C07280=1077.683,437.352,387.565,177.005,33.132,155.992
C07281=1077.692,437.598,387.519,177.011,33.146,155.996
C07282=1077.700,437.843,387.473,177.017,33.159,155.999
C07283=1077.707,438.089,387.426,177.024,33.173,156.002
C07284=1077.715,438.334,387.380,177.031,33.186,156.005
C07285=1077.726,438.676,387.315,177.040,33.205,156.010
C07286=1077.738,439.018,387.250,177.048,33.224,156.014
C07287=1077.749,439.359,387.186,177.058,33.243,156.019
C07288=1077.761,439.701,387.121,177.067,33.262,156.023
C07289=1077.771,440.033,387.057,177.077,33.281,156.028
C07290=1077.782,440.366,386.995,177.085,33.300,156.032
C07291=1077.793,440.699,386.931,177.094,33.319,156.037
C07292=1077.804,441.033,386.867,177.104,33.338,156.041
C07293=1077.812,441.277,386.821,177.110,33.352,156.045
C07294=1077.820,441.523,386.774,177.118,33.366,156.048
C07295=1077.829,441.768,386.726,177.124,33.380,156.052
C07296=1077.837,442.014,386.679,177.130,33.395,156.055
C07297=1077.845,442.259,386.633,177.138,33.409,156.059
C07298=1077.853,442.504,386.584,177.144,33.423,156.062
C07299=1077.861,442.749,386.538,177.152,33.438,156.065
C07300=1077.869,442.995,386.490,177.158,33.452,156.069
C07301=1077.877,443.239,386.443,177.166,33.467,156.072
C07302=1077.885,443.485,386.396,177.173,33.482,156.076
C07303=1077.894,443.730,386.349,177.179,33.496,156.080
C07304=1077.902,443.976,386.301,177.187,33.511,156.083
C07305=1077.911,444.221,386.254,177.193,33.525,156.087
C07306=1077.919,444.467,386.206,177.201,33.540,156.090
C07307=1077.927,444.712,386.158,177.208,33.555,156.094
C07308=1077.935,444.957,386.111,177.215,33.570,156.097
C07309=1077.944,445.202,386.063,177.222,33.585,156.101
C07310=1077.952,445.447,386.015,177.229,33.600,156.105
C07311=1077.960,445.693,385.968,177.237,33.615,156.108
C07312=1077.968,445.938,385.920,177.244,33.630,156.112
C07313=1077.976,446.183,385.872,177.252,33.645,156.116
C07314=1077.985,446.428,385.825,177.258,33.660,156.119
C07315=1077.993,446.673,385.777,177.265,33.675,156.123
C07316=1078.002,446.918,385.729,177.271,33.690,156.127
C07317=1078.010,447.164,385.681,177.278,33.706,156.131
C07318=1078.019,447.408,385.632,177.285,33.721,156.134
C07319=1078.027,447.653,385.584,177.290,33.736,156.138
C07320=1078.035,447.898,385.536,177.296,33.751,156.142
C07321=1078.043,448.143,385.488,177.302,33.766,156.146
C07322=1078.052,448.388,385.440,177.306,33.781,156.149
C07323=1078.061,448.634,385.392,177.311,33.796,156.153
C07324=1078.069,448.878,385.343,177.316,33.811,156.157
C07325=1078.079,449.123,385.296,177.320,33.826,156.161
C07326=1078.090,449.368,385.249,177.325,33.840,156.164
C07327=1078.102,449.613,385.203,177.329,33.853,156.168
C07328=1078.116,449.859,385.158,177.333,33.866,156.171
C07329=1077.755,449.854,384.928,177.311,34.027,156.213
C07330=1077.741,449.608,384.974,177.306,34.015,156.210
C07331=1077.728,449.363,385.020,177.302,34.001,156.207
C07332=1077.716,449.117,385.067,177.298,33.987,156.203
C07333=1077.707,448.873,385.113,177.293,33.973,156.200
C07334=1077.698,448.628,385.162,177.288,33.958,156.196
C07335=1077.690,448.383,385.210,177.283,33.942,156.192
C07336=1077.681,448.139,385.258,177.277,33.927,156.188
C07337=1077.673,447.894,385.306,177.272,33.912,156.185
C07338=1077.664,447.649,385.355,177.266,33.897,156.181
C07339=1077.656,447.403,385.404,177.260,33.882,156.177
C07340=1077.647,447.158,385.451,177.253,33.867,156.173
C07341=1077.639,446.913,385.499,177.248,33.852,156.170
C07342=1077.631,446.668,385.547,177.240,33.836,156.166
C07343=1077.622,446.423,385.596,177.233,33.821,156.162
C07344=1077.613,446.178,385.643,177.226,33.806,156.158
C07345=1077.605,445.933,385.691,177.219,33.791,156.155
C07346=1077.597,445.688,385.739,177.211,33.776,156.151
C07347=1077.589,445.443,385.787,177.204,33.761,156.147
C07348=1077.580,445.198,385.835,177.197,33.746,156.144
C07349=1077.572,444.952,385.882,177.189,33.731,156.140
C07350=1077.564,444.707,385.930,177.182,33.716,156.136
C07351=1077.555,444.462,385.978,177.175,33.701,156.133
C07352=1077.547,444.217,386.026,177.168,33.686,156.129
C07353=1077.539,443.971,386.072,177.161,33.672,156.126
C07354=1077.531,443.726,386.120,177.153,33.657,156.122
C07355=1077.522,443.481,386.168,177.146,33.643,156.118
C07356=1077.514,443.235,386.215,177.139,33.628,156.115
C07357=1077.506,442.990,386.263,177.132,33.613,156.111
C07358=1077.497,442.745,386.310,177.125,33.599,156.108
C07359=1077.490,442.500,386.358,177.118,33.585,156.104
C07360=1077.481,442.255,386.404,177.111,33.570,156.101
C07361=1077.474,442.009,386.452,177.104,33.556,156.097
C07362=1077.465,441.764,386.499,177.097,33.542,156.094
C07363=1077.457,441.519,386.546,177.090,33.527,156.091
C07364=1077.449,441.273,386.593,177.083,33.513,156.087
C07365=1077.440,441.028,386.640,177.077,33.499,156.084
C07366=1077.430,440.712,386.700,177.067,33.481,156.079
C07367=1077.420,440.397,386.761,177.059,33.463,156.075
C07368=1077.409,440.080,386.821,177.050,33.445,156.071
C07369=1077.399,439.764,386.881,177.042,33.427,156.067
C07370=1077.391,439.519,386.928,177.034,33.413,156.063
C07371=1077.383,439.274,386.975,177.028,33.399,156.060
C07372=1077.375,439.029,387.021,177.022,33.386,156.057
C07373=1077.367,438.783,387.067,177.014,33.372,156.053
C07374=1077.358,438.537,387.114,177.008,33.359,156.050
C07375=1077.350,438.292,387.161,177.002,33.345,156.047
C07376=1077.342,438.046,387.207,176.994,33.332,156.044
C07377=1077.334,437.801,387.253,176.988,33.318,156.040
C07378=1077.326,437.555,387.300,176.982,33.305,156.037
C07379=1077.319,437.310,387.346,176.975,33.291,156.034
C07380=1077.310,437.065,387.393,176.968,33.278,156.031
C07381=1077.302,436.819,387.438,176.962,33.265,156.028
C07382=1077.294,436.574,387.485,176.955,33.251,156.025
C07383=1077.286,436.328,387.531,176.949,33.238,156.021
C07384=1077.278,436.082,387.577,176.943,33.225,156.018
C07385=1077.270,435.837,387.623,176.936,33.212,156.015
C07386=1077.262,435.592,387.669,176.929,33.199,156.012
C07387=1077.254,435.346,387.715,176.923,33.186,156.009
C07388=1077.246,435.101,387.761,176.917,33.173,156.006
C07389=1077.239,434.855,387.807,176.911,33.160,156.003
C07390=1077.230,434.609,387.853,176.904,33.147,156.000
C07391=1077.223,434.364,387.898,176.898,33.134,155.997
C07392=1077.215,434.118,387.944,176.892,33.121,155.994
C07393=1077.207,433.872,387.990,176.886,33.108,155.991
C07394=1077.200,433.627,388.036,176.880,33.095,155.988
C07395=1077.192,433.381,388.082,176.872,33.083,155.985
C07396=1077.184,433.136,388.127,176.866,33.070,155.982
C07397=1077.176,432.891,388.173,176.860,33.058,155.979
C07398=1077.168,432.644,388.219,176.854,33.045,155.976
C07399=1077.161,432.398,388.264,176.848,33.032,155.973
C07400=1077.153,432.153,388.309,176.842,33.020,155.970
C07401=1077.145,431.907,388.355,176.835,33.007,155.967
C07402=1077.138,431.662,388.401,176.829,32.995,155.964
C07403=1077.130,431.416,388.445,176.824,32.982,155.961
C07404=1077.122,431.170,388.491,176.818,32.970,155.958
C07405=1077.114,430.924,388.536,176.812,32.958,155.956
C07406=1077.107,430.679,388.581,176.806,32.946,155.953
C07407=1077.099,430.433,388.626,176.800,32.933,155.950
C07408=1077.091,430.187,388.671,176.794,32.921,155.947
C07409=1077.083,429.941,388.716,176.788,32.909,155.944
C07410=1077.076,429.696,388.762,176.781,32.897,155.941
C07411=1077.069,429.450,388.807,176.775,32.885,155.939
C07412=1077.060,429.204,388.851,176.769,32.873,155.936
C07413=1077.053,428.959,388.897,176.763,32.861,155.933
C07414=1077.045,428.713,388.942,176.758,32.849,155.930
C07415=1077.037,428.467,388.986,176.752,32.837,155.928
C07416=1077.030,428.221,389.031,176.746,32.825,155.925
C07417=1077.023,427.975,389.076,176.740,32.813,155.922
C07418=1077.013,427.678,389.130,176.733,32.799,155.919
C07419=1077.004,427.380,389.184,176.726,32.785,155.916
C07420=1076.994,427.083,389.238,176.719,32.770,155.912
C07421=1076.986,426.787,389.292,176.712,32.756,155.909
C07422=1076.978,426.571,389.331,176.707,32.747,155.907
C07423=1076.972,426.356,389.370,176.702,32.737,155.904
C07424=1076.965,426.141,389.409,176.697,32.726,155.902
C07425=1076.959,425.925,389.447,176.692,32.716,155.900
C07426=1076.951,425.680,389.492,176.686,32.705,155.897
C07427=1076.944,425.433,389.537,176.681,32.693,155.894
C07428=1076.936,425.188,389.581,176.675,32.682,155.892
C07429=1076.929,424.941,389.625,176.669,32.671,155.889
C07430=1076.921,424.696,389.669,176.664,32.659,155.887
C07431=1076.913,424.450,389.713,176.658,32.648,155.884
C07432=1076.906,424.204,389.758,176.652,32.637,155.881
C07433=1076.898,423.958,389.802,176.647,32.625,155.879
C07434=1076.892,423.712,389.846,176.641,32.614,155.876
C07435=1076.884,423.466,389.890,176.635,32.603,155.874
C07436=1076.876,423.220,389.934,176.630,32.592,155.871
C07437=1076.869,422.974,389.978,176.625,32.581,155.869
C07438=1076.861,422.728,390.022,176.620,32.569,155.866
C07439=1076.854,422.482,390.067,176.614,32.559,155.864
C07440=1076.847,422.236,390.110,176.608,32.547,155.861
C07441=1076.839,421.990,390.154,176.603,32.536,155.859
C07442=1076.832,421.745,390.198,176.597,32.525,155.856
C07443=1076.825,421.498,390.242,176.592,32.515,155.854
C07444=1076.817,421.252,390.286,176.586,32.504,155.851
C07445=1076.810,421.006,390.329,176.581,32.493,155.849
C07446=1076.802,420.760,390.372,176.575,32.482,155.846
C07447=1076.794,420.513,390.416,176.570,32.472,155.844
C07448=1076.787,420.268,390.459,176.565,32.461,155.841
C07449=1076.780,420.021,390.504,176.560,32.450,155.839
C07450=1076.773,419.775,390.547,176.554,32.439,155.837
C07451=1076.765,419.529,390.590,176.549,32.428,155.834
C07452=1076.758,419.283,390.634,176.543,32.418,155.832
C07453=1076.750,419.037,390.677,176.538,32.408,155.830
C07454=1076.743,418.791,390.721,176.532,32.397,155.827
C07455=1076.735,418.545,390.764,176.528,32.386,155.825
C07456=1076.728,418.299,390.807,176.522,32.376,155.822
C07457=1076.720,418.053,390.851,176.517,32.366,155.820
C07458=1076.713,417.807,390.894,176.512,32.355,155.818
C07459=1076.706,417.561,390.937,176.506,32.345,155.815
C07460=1076.698,417.315,390.980,176.501,32.334,155.813
C07461=1076.692,417.068,391.023,176.496,32.324,155.811
C07462=1076.684,416.822,391.067,176.491,32.314,155.808
C07463=1076.677,416.576,391.110,176.486,32.303,155.806
C07464=1076.670,416.330,391.152,176.480,32.293,155.804
C07465=1076.662,416.084,391.196,176.475,32.283,155.802
C07466=1076.655,415.837,391.239,176.470,32.272,155.799
C07467=1076.648,415.592,391.282,176.465,32.262,155.797
C07468=1076.641,415.346,391.324,176.460,32.252,155.795
C07469=1076.634,415.099,391.367,176.455,32.242,155.792
C07470=1076.627,414.853,391.411,176.449,32.232,155.790
C07471=1076.619,414.607,391.452,176.444,32.222,155.788
C07472=1076.611,414.360,391.495,176.440,32.212,155.786
C07473=1076.604,414.114,391.539,176.435,32.203,155.784
C07474=1076.597,413.868,391.581,176.429,32.193,155.781
C07475=1076.589,413.621,391.623,176.424,32.183,155.779
C07476=1076.582,413.375,391.666,176.420,32.173,155.777
C07477=1076.576,413.129,391.709,176.414,32.163,155.775
C07478=1076.569,412.880,391.752,176.409,32.153,155.773
C07479=1076.560,412.631,391.795,176.404,32.143,155.770
C07480=1076.553,412.382,391.838,176.399,32.133,155.768
C07481=1076.546,412.132,391.881,176.394,32.123,155.766
C07482=1076.539,411.886,391.923,176.389,32.114,155.764
C07483=1076.531,411.640,391.965,176.384,32.104,155.762
C07484=1076.525,411.394,392.008,176.379,32.094,155.760
C07485=1076.518,411.148,392.050,176.375,32.085,155.758
C07486=1076.510,410.902,392.092,176.369,32.075,155.755
C07487=1076.503,410.655,392.135,176.364,32.065,155.753
C07488=1076.496,410.409,392.177,176.359,32.056,155.751
C07489=1076.489,410.162,392.218,176.355,32.047,155.749
C07490=1076.482,409.915,392.261,176.350,32.037,155.747
C07491=1076.474,409.669,392.303,176.345,32.027,155.745
C07492=1076.467,409.423,392.346,176.341,32.018,155.743
C07493=1076.461,409.176,392.388,176.336,32.008,155.741
C07494=1076.453,408.930,392.430,176.330,31.999,155.739
C07495=1076.447,408.685,392.472,176.325,31.989,155.737
C07496=1076.440,408.438,392.513,176.321,31.981,155.735
C07497=1076.433,408.192,392.556,176.316,31.971,155.733
C07498=1076.425,407.946,392.597,176.311,31.962,155.731
C07499=1076.419,407.699,392.639,176.307,31.952,155.729
C07500=1076.412,407.453,392.682,176.302,31.943,155.727
C07501=1076.404,407.206,392.723,176.297,31.934,155.725
C07502=1076.398,406.959,392.765,176.292,31.925,155.723
C07503=1076.390,406.713,392.807,176.288,31.915,155.721
C07504=1076.384,406.466,392.849,176.283,31.907,155.719
C07505=1076.376,406.220,392.891,176.278,31.897,155.717
C07506=1076.369,405.974,392.931,176.274,31.888,155.715
C07507=1076.363,405.727,392.973,176.269,31.879,155.713
C07508=1076.356,405.481,393.015,176.264,31.870,155.711
C07509=1076.348,405.235,393.056,176.260,31.861,155.709
C07510=1076.341,404.988,393.098,176.255,31.852,155.707
C07511=1076.334,404.741,393.140,176.250,31.843,155.705
C07512=1076.327,404.496,393.180,176.246,31.834,155.703
C07513=1076.321,404.249,393.222,176.241,31.825,155.701
C07514=1076.313,404.003,393.264,176.236,31.817,155.699
C07515=1076.306,403.756,393.305,176.232,31.808,155.697
C07516=1076.300,403.510,393.347,176.227,31.799,155.695
C07517=1076.293,403.263,393.388,176.222,31.790,155.693
C07518=1076.286,403.017,393.429,176.219,31.781,155.691
C07519=1076.278,402.770,393.471,176.214,31.772,155.690
C07520=1076.272,402.524,393.511,176.209,31.764,155.688
C07521=1076.265,402.277,393.552,176.205,31.755,155.686
C07522=1076.257,402.030,393.593,176.200,31.746,155.684
C07523=1076.251,401.784,393.635,176.195,31.738,155.682
C07524=1076.244,401.538,393.676,176.191,31.729,155.680
C07525=1076.237,401.291,393.717,176.186,31.720,155.678
C07526=1076.230,401.045,393.758,176.181,31.712,155.677
C07527=1076.223,400.798,393.798,176.178,31.703,155.675
C07528=1076.216,400.551,393.840,176.173,31.695,155.673
C07529=1076.209,400.305,393.881,176.168,31.686,155.671
C07530=1076.202,400.059,393.922,176.164,31.678,155.669
C07531=1076.195,399.812,393.962,176.159,31.669,155.667
C07532=1076.188,399.566,394.003,176.154,31.661,155.666
C07533=1076.181,399.320,394.044,176.151,31.652,155.664
C07534=1076.175,399.074,394.085,176.146,31.644,155.662
C07535=1076.168,398.827,394.125,176.142,31.635,155.660
C07536=1076.161,398.581,394.166,176.137,31.627,155.658
C07537=1076.155,398.334,394.206,176.132,31.619,155.657
C07538=1076.147,398.088,394.248,176.129,31.611,155.655
C07539=1076.141,397.841,394.288,176.124,31.602,155.653
C07540=1076.134,397.595,394.329,176.119,31.594,155.651
C07541=1076.127,397.348,394.369,176.115,31.586,155.650
C07542=1076.119,397.102,394.410,176.111,31.578,155.648
C07543=1076.113,396.855,394.450,176.107,31.569,155.646
C07544=1076.106,396.608,394.490,176.102,31.561,155.644
C07545=1076.099,396.362,394.531,176.097,31.553,155.643
C07546=1076.092,396.115,394.572,176.094,31.545,155.641
C07547=1076.086,395.868,394.612,176.089,31.537,155.639
C07548=1076.079,395.622,394.651,176.084,31.528,155.638
C07549=1076.072,395.376,394.693,176.080,31.520,155.636
C07550=1076.065,395.129,394.733,176.076,31.512,155.634
C07551=1076.059,394.883,394.773,176.072,31.504,155.632
C07552=1076.052,394.635,394.814,176.067,31.496,155.631
C07553=1076.045,394.389,394.853,176.063,31.489,155.629
C07554=1076.038,394.143,394.893,176.059,31.481,155.627
C07555=1076.031,393.895,394.934,176.054,31.472,155.626
C07556=1076.025,393.649,394.974,176.050,31.464,155.624
C07557=1076.018,393.403,395.013,176.046,31.457,155.622
C07558=1076.011,393.155,395.054,176.041,31.449,155.621
C07559=1076.004,392.909,395.094,176.037,31.441,155.619
C07560=1075.997,392.663,395.134,176.033,31.433,155.617
C07561=1075.991,392.416,395.174,176.029,31.425,155.616
C07562=1075.983,392.169,395.214,176.024,31.417,155.614
C07563=1075.977,391.923,395.254,176.020,31.409,155.612
C07564=1075.971,391.676,395.294,176.016,31.402,155.611
C07565=1075.963,391.430,395.334,176.011,31.394,155.609
C07566=1075.957,391.183,395.373,176.008,31.386,155.608
C07567=1075.950,390.936,395.413,176.003,31.378,155.606
C07568=1075.943,390.690,395.453,175.999,31.371,155.604
C07569=1075.936,390.443,395.493,175.995,31.363,155.603
C07570=1075.930,390.196,395.532,175.990,31.355,155.601
C07571=1075.923,389.950,395.572,175.986,31.348,155.600
C07572=1075.915,389.702,395.611,175.982,31.340,155.598
C07573=1075.909,389.456,395.651,175.978,31.332,155.596
C07574=1075.902,389.210,395.691,175.974,31.325,155.595
C07575=1075.896,388.963,395.730,175.970,31.317,155.593
C07576=1075.889,388.716,395.769,175.965,31.310,155.592
C07577=1075.882,388.470,395.808,175.961,31.302,155.590
C07578=1075.876,388.223,395.848,175.957,31.295,155.589
C07579=1075.869,387.976,395.887,175.953,31.287,155.587
C07580=1075.862,387.730,395.927,175.949,31.280,155.586
C07581=1075.856,387.483,395.966,175.944,31.272,155.584
C07582=1075.848,387.237,396.006,175.941,31.265,155.583
C07583=1075.841,386.989,396.045,175.936,31.257,155.581
C07584=1075.835,386.742,396.084,175.932,31.250,155.579
C07585=1075.828,386.496,396.124,175.928,31.243,155.578
C07586=1075.822,386.257,396.161,175.924,31.236,155.576
C07587=1075.816,386.018,396.200,175.920,31.228,155.575
C07588=1075.809,385.779,396.237,175.916,31.222,155.574
C07589=1075.803,385.540,396.275,175.913,31.214,155.572
C07590=1075.796,385.301,396.314,175.908,31.207,155.571
C07591=1075.790,385.062,396.352,175.904,31.200,155.569
C07592=1075.784,384.824,396.389,175.900,31.193,155.568
C07593=1075.777,384.585,396.427,175.896,31.186,155.566
C07594=1075.770,384.338,396.466,175.893,31.179,155.565
C07595=1075.764,384.091,396.505,175.888,31.171,155.563
C07596=1075.757,383.844,396.545,175.885,31.164,155.562
C07597=1075.751,383.598,396.583,175.880,31.157,155.560
C07598=1075.744,383.351,396.622,175.876,31.150,155.559
C07599=1075.738,383.104,396.661,175.872,31.142,155.557
C07600=1075.731,382.857,396.700,175.868,31.135,155.556
C07601=1075.724,382.611,396.739,175.864,31.128,155.555
C07602=1075.717,382.364,396.778,175.860,31.121,155.553
C07603=1075.711,382.117,396.817,175.856,31.114,155.552
C07604=1075.705,381.870,396.855,175.852,31.107,155.550
C07605=1075.699,381.623,396.894,175.848,31.100,155.549
C07606=1075.692,381.376,396.933,175.844,31.093,155.547
C07607=1075.685,381.129,396.972,175.840,31.086,155.546
C07608=1075.678,380.883,397.011,175.836,31.079,155.544
C07609=1075.672,380.635,397.049,175.831,31.072,155.543
C07610=1075.665,380.389,397.087,175.828,31.065,155.542
C07611=1075.659,380.142,397.126,175.824,31.058,155.540
C07612=1075.652,379.895,397.165,175.820,31.051,155.539
C07613=1075.645,379.648,397.203,175.816,31.044,155.537
C07614=1075.638,379.401,397.241,175.812,31.037,155.536
C07615=1075.632,379.155,397.280,175.808,31.030,155.535
C07616=1075.625,378.908,397.318,175.804,31.023,155.533
C07617=1075.618,378.661,397.357,175.800,31.016,155.532
C07618=1075.612,378.414,397.395,175.797,31.010,155.531
C07619=1075.606,378.168,397.433,175.792,31.003,155.529
C07620=1075.599,377.920,397.471,175.789,30.996,155.528
C07621=1075.592,377.673,397.510,175.784,30.989,155.526
C07622=1075.586,377.426,397.548,175.781,30.982,155.525
C07623=1075.579,377.180,397.587,175.777,30.975,155.524
C07624=1075.573,376.932,397.625,175.772,30.969,155.522
C07625=1075.566,376.686,397.663,175.769,30.962,155.521
C07626=1075.560,376.439,397.701,175.765,30.955,155.520
C07627=1075.553,376.192,397.739,175.761,30.948,155.518
C07628=1075.547,375.945,397.777,175.757,30.942,155.517
C07629=1075.540,375.698,397.816,175.754,30.935,155.516
C07630=1075.534,375.450,397.854,175.749,30.928,155.514
C07631=1075.528,375.204,397.892,175.746,30.922,155.513
C07632=1075.521,374.957,397.930,175.741,30.915,155.511
C07633=1075.514,374.711,397.967,175.738,30.908,155.510
C07634=1075.508,374.463,398.006,175.734,30.902,155.509
C07635=1075.502,374.217,398.044,175.730,30.895,155.507
C07636=1075.495,373.969,398.082,175.726,30.888,155.506
C07637=1075.489,373.722,398.120,175.723,30.882,155.505
C07638=1075.483,373.475,398.158,175.719,30.875,155.504
C07639=1075.476,373.228,398.196,175.715,30.869,155.502
C07640=1075.470,372.981,398.233,175.711,30.862,155.501
C07641=1075.462,372.734,398.271,175.708,30.856,155.500
C07642=1075.456,372.510,398.306,175.704,30.850,155.499
C07643=1075.451,372.285,398.340,175.700,30.844,155.497
C07644=1075.445,372.062,398.374,175.697,30.838,155.496
C07645=1075.439,371.837,398.408,175.693,30.832,155.495
C07646=1075.433,371.612,398.443,175.690,30.826,155.494
C07647=1075.427,371.388,398.476,175.686,30.820,155.493
C07648=1075.421,371.164,398.511,175.683,30.815,155.492
C07649=1075.416,370.939,398.545,175.679,30.809,155.490
C07650=1075.408,370.692,398.582,175.676,30.802,155.489
C07651=1075.402,370.445,398.620,175.672,30.796,155.488
C07652=1075.395,370.198,398.657,175.668,30.790,155.487
C07653=1075.390,369.951,398.695,175.664,30.783,155.485
C07654=1075.383,369.704,398.733,175.660,30.777,155.484
C07655=1075.376,369.457,398.770,175.657,30.770,155.483
C07656=1075.370,369.210,398.808,175.652,30.764,155.482
C07657=1075.364,368.963,398.844,175.649,30.758,155.480
C07658=1075.358,368.716,398.882,175.645,30.752,155.479
C07659=1075.350,368.469,398.920,175.642,30.745,155.478
C07660=1075.345,368.221,398.957,175.638,30.739,155.477
C07661=1075.338,367.974,398.994,175.634,30.733,155.476
C07662=1075.332,367.727,399.032,175.630,30.726,155.474
C07663=1075.325,367.480,399.068,175.627,30.720,155.473
C07664=1075.318,367.233,399.106,175.623,30.714,155.472
C07665=1075.313,366.986,399.143,175.619,30.708,155.471
C07666=1075.306,366.740,399.180,175.615,30.701,155.469
C07667=1075.300,366.491,399.218,175.612,30.695,155.468
C07668=1075.293,366.245,399.255,175.608,30.689,155.467
C07669=1075.287,365.998,399.292,175.605,30.683,155.466
C07670=1075.280,365.750,399.329,175.600,30.677,155.465
C07671=1075.275,365.503,399.366,175.597,30.671,155.463
C07672=1075.268,365.257,399.403,175.593,30.664,155.462
C07673=1075.262,365.010,399.440,175.590,30.658,155.461
C07674=1075.255,364.762,399.477,175.586,30.652,155.460
C07675=1075.249,364.515,399.514,175.582,30.646,155.459
C07676=1075.242,364.268,399.551,175.578,30.640,155.457
C07677=1075.236,364.020,399.588,175.575,30.634,155.456
C07678=1075.230,363.773,399.625,175.571,30.628,155.455
C07679=1075.223,363.527,399.662,175.568,30.622,155.454
C07680=1075.217,363.279,399.698,175.564,30.616,155.453
C07681=1075.210,363.032,399.735,175.560,30.610,155.452
C07682=1075.204,362.784,399.772,175.556,30.604,155.450
C07683=1075.198,362.537,399.809,175.553,30.598,155.449
C07684=1075.191,362.291,399.846,175.549,30.592,155.448
C07685=1075.184,362.043,399.883,175.546,30.586,155.447
C07686=1075.178,361.796,399.919,175.542,30.580,155.446
C07687=1075.172,361.549,399.956,175.539,30.574,155.445
C07688=1075.165,361.302,399.992,175.534,30.568,155.444
C07689=1075.160,361.055,400.029,175.531,30.562,155.442
C07690=1075.153,360.807,400.066,175.527,30.556,155.441
C07691=1075.147,360.560,400.102,175.524,30.550,155.440
C07692=1075.140,360.313,400.139,175.520,30.545,155.439
C07693=1075.134,360.066,400.175,175.517,30.539,155.438
C07694=1075.128,359.819,400.212,175.513,30.533,155.437
C07695=1075.121,359.572,400.248,175.510,30.527,155.436
C07696=1075.115,359.325,400.285,175.505,30.521,155.435
C07697=1075.108,359.076,400.321,175.502,30.515,155.433
C07698=1075.103,358.861,400.352,175.499,30.510,155.432
C07699=1075.097,358.645,400.384,175.496,30.505,155.431
C07700=1075.092,358.428,400.416,175.493,30.500,155.430
C07701=1075.086,358.212,400.448,175.490,30.495,155.430
C07702=1075.080,357.996,400.480,175.486,30.490,155.429
C07703=1075.075,357.780,400.511,175.483,30.485,155.428
C07704=1075.070,357.564,400.543,175.480,30.480,155.427
C07705=1075.064,357.348,400.575,175.477,30.475,155.426
C07706=1075.057,357.101,400.611,175.474,30.469,155.425
C07707=1075.051,356.853,400.647,175.470,30.463,155.423
C07708=1075.045,356.606,400.683,175.466,30.457,155.422
C07709=1075.039,356.359,400.720,175.462,30.452,155.421
C07710=1075.033,356.111,400.756,175.459,30.446,155.420
C07711=1075.026,355.864,400.792,175.455,30.440,155.419
C07712=1075.020,355.617,400.828,175.452,30.434,155.418
C07713=1075.014,355.369,400.864,175.448,30.429,155.417
C07714=1075.008,355.122,400.901,175.445,30.423,155.416
C07715=1075.002,354.875,400.936,175.441,30.417,155.415
C07716=1074.995,354.628,400.972,175.438,30.412,155.414
C07717=1074.989,354.380,401.008,175.434,30.406,155.413
C07718=1074.982,354.133,401.044,175.431,30.401,155.412
C07719=1074.976,353.886,401.080,175.427,30.395,155.411
C07720=1074.970,353.638,401.116,175.424,30.389,155.409
C07721=1074.964,353.391,401.152,175.420,30.384,155.408
C07722=1074.958,353.143,401.188,175.417,30.378,155.407
C07723=1074.951,352.896,401.224,175.413,30.372,155.406
C07724=1074.945,352.649,401.260,175.410,30.367,155.405
C07725=1074.939,352.401,401.295,175.406,30.361,155.404
C07726=1074.932,352.154,401.332,175.403,30.356,155.403
C07727=1074.926,351.907,401.367,175.400,30.350,155.402
C07728=1074.920,351.659,401.403,175.396,30.345,155.401
C07729=1074.913,351.411,401.438,175.393,30.339,155.400
C07730=1074.906,351.165,401.474,175.389,30.334,155.399
C07731=1074.901,350.918,401.510,175.386,30.328,155.398
C07732=1074.895,350.670,401.545,175.382,30.323,155.397
C07733=1074.888,350.423,401.580,175.379,30.317,155.396
C07734=1074.882,350.175,401.616,175.375,30.312,155.395
C07735=1074.876,349.927,401.652,175.372,30.306,155.394
C07736=1074.869,349.681,401.688,175.368,30.301,155.393
C07737=1074.863,349.433,401.723,175.365,30.296,155.392
C07738=1074.856,349.185,401.759,175.361,30.290,155.391
C07739=1074.851,348.938,401.794,175.358,30.285,155.390
C07740=1074.845,348.691,401.830,175.354,30.279,155.389
C07741=1074.838,348.443,401.865,175.351,30.274,155.388
C07742=1074.832,348.196,401.901,175.347,30.269,155.387
C07743=1074.825,347.948,401.936,175.344,30.263,155.386
C07744=1074.820,347.701,401.971,175.340,30.258,155.385
C07745=1074.813,347.454,402.006,175.337,30.252,155.384
C07746=1074.807,347.206,402.042,175.333,30.247,155.383
C07747=1074.801,346.958,402.076,175.330,30.242,155.382
C07748=1074.795,346.711,402.112,175.326,30.236,155.381
C07749=1074.789,346.464,402.147,175.323,30.231,155.380
C07750=1074.782,346.216,402.183,175.320,30.226,155.379
C07751=1074.776,345.969,402.218,175.317,30.220,155.378
C07752=1074.770,345.721,402.253,175.313,30.215,155.377
C07753=1074.763,345.475,402.288,175.310,30.210,155.376
C07754=1074.758,345.260,402.318,175.306,30.205,155.375
C07755=1074.753,345.045,402.349,175.304,30.200,155.374
C07756=1074.748,344.831,402.379,175.301,30.196,155.373
C07757=1074.742,344.616,402.410,175.298,30.191,155.373
C07758=1074.737,344.402,402.441,175.295,30.187,155.372
C07759=1074.731,344.188,402.471,175.293,30.182,155.371
C07760=1074.726,343.974,402.501,175.289,30.178,155.370
C07761=1074.721,343.759,402.531,175.286,30.173,155.369
C07762=1074.714,343.511,402.566,175.283,30.168,155.368
C07763=1074.708,343.265,402.601,175.279,30.163,155.367
C07764=1074.702,343.016,402.636,175.276,30.158,155.366
C07765=1074.695,342.769,402.671,175.273,30.152,155.365
C07766=1074.690,342.522,402.705,175.269,30.147,155.364
C07767=1074.684,342.274,402.741,175.266,30.142,155.363
C07768=1074.677,342.026,402.775,175.263,30.137,155.362
C07769=1074.671,341.779,402.810,175.260,30.132,155.362
C07770=1074.664,341.531,402.845,175.256,30.126,155.361
C07771=1074.658,341.284,402.880,175.253,30.121,155.360
C07772=1074.653,341.036,402.914,175.249,30.116,155.359
C07773=1074.646,340.789,402.950,175.246,30.111,155.358
C07774=1074.640,340.542,402.984,175.242,30.105,155.357
C07775=1074.634,340.294,403.019,175.239,30.100,155.356
C07776=1074.627,340.046,403.054,175.236,30.096,155.355
C07777=1074.622,339.799,403.088,175.233,30.091,155.354
C07778=1074.615,339.551,403.123,175.229,30.085,155.353
C07779=1074.609,339.304,403.157,175.226,30.080,155.352
C07780=1074.603,339.056,403.192,175.222,30.075,155.351
C07781=1074.597,338.808,403.226,175.219,30.070,155.350
C07782=1074.591,338.561,403.261,175.216,30.065,155.349
C07783=1074.585,338.314,403.295,175.213,30.060,155.348
C07784=1074.578,338.066,403.330,175.209,30.055,155.348
C07785=1074.573,337.818,403.364,175.206,30.049,155.347
C07786=1074.566,337.571,403.399,175.202,30.044,155.346
C07787=1074.560,337.323,403.434,175.200,30.040,155.345
C07788=1074.554,337.076,403.468,175.196,30.035,155.344
C07789=1074.548,336.828,403.502,175.193,30.030,155.343
C07790=1074.542,336.580,403.536,175.189,30.024,155.342
C07791=1074.535,336.332,403.571,175.186,30.019,155.341
C07792=1074.529,336.085,403.605,175.183,30.014,155.340
C07793=1074.523,335.837,403.639,175.180,30.010,155.339
C07794=1074.517,335.590,403.673,175.177,30.004,155.338
C07795=1074.511,335.342,403.708,175.173,29.999,155.338
C07796=1074.504,335.095,403.742,175.170,29.994,155.337
C07797=1074.498,334.847,403.776,175.167,29.990,155.336
C07798=1074.492,334.600,403.810,175.164,29.985,155.335
C07799=1074.486,334.352,403.844,175.160,29.980,155.334
C07800=1074.479,334.104,403.878,175.157,29.975,155.333
C07801=1074.474,333.857,403.912,175.153,29.970,155.332
C07802=1074.467,333.609,403.947,175.151,29.965,155.331
C07803=1074.461,333.362,403.981,175.147,29.960,155.330
C07804=1074.455,333.114,404.015,175.144,29.955,155.330
C07805=1074.449,332.866,404.049,175.140,29.950,155.329
C07806=1074.443,332.619,404.083,175.138,29.946,155.328
C07807=1074.437,332.371,404.117,175.134,29.940,155.327
C07808=1074.431,332.123,404.151,175.131,29.935,155.326
C07809=1074.425,331.876,404.185,175.127,29.930,155.325
C07810=1074.419,331.659,404.215,175.125,29.926,155.324
C07811=1074.414,331.443,404.244,175.122,29.922,155.324
C07812=1074.408,331.225,404.274,175.120,29.918,155.323
C07813=1074.403,331.009,404.303,175.116,29.913,155.322
C07814=1074.398,330.791,404.334,175.114,29.910,155.321
C07815=1074.392,330.573,404.363,175.111,29.905,155.321
C07816=1074.387,330.357,404.393,175.108,29.901,155.320
C07817=1074.381,330.140,404.422,175.105,29.897,155.319
C07818=1074.375,329.892,404.455,175.102,29.892,155.318
C07819=1074.369,329.644,404.490,175.099,29.888,155.318
C07820=1074.362,329.397,404.522,175.096,29.882,155.317
C07821=1074.356,329.150,404.556,175.092,29.878,155.316
C07822=1074.350,328.902,404.591,175.090,29.873,155.315
C07823=1074.344,328.654,404.624,175.086,29.868,155.314
C07824=1074.338,328.407,404.658,175.083,29.863,155.313
C07825=1074.331,328.158,404.691,175.079,29.859,155.312
C07826=1074.325,327.911,404.725,175.077,29.854,155.312
C07827=1074.319,327.663,404.758,175.073,29.849,155.311
C07828=1074.312,327.415,404.792,175.070,29.844,155.310
C07829=1074.306,327.168,404.825,175.067,29.840,155.309
C07830=1074.300,326.920,404.858,175.064,29.835,155.308
C07831=1074.295,326.673,404.892,175.060,29.830,155.307
C07832=1074.288,326.424,404.925,175.057,29.826,155.307
C07833=1074.282,326.177,404.959,175.054,29.821,155.306
C07834=1074.276,325.930,404.992,175.051,29.816,155.305
C07835=1074.270,325.682,405.025,175.047,29.811,155.304
C07836=1074.263,325.434,405.059,175.045,29.807,155.303
C07837=1074.257,325.186,405.092,175.041,29.802,155.303
C07838=1074.251,324.938,405.125,175.038,29.797,155.302
C07839=1074.245,324.691,405.159,175.035,29.793,155.301
C07840=1074.239,324.444,405.192,175.032,29.788,155.300
C07841=1074.233,324.195,405.226,175.028,29.783,155.299
C07842=1074.226,323.947,405.258,175.026,29.779,155.298
C07843=1074.221,323.699,405.292,175.022,29.774,155.298
C07844=1074.214,323.453,405.325,175.020,29.770,155.297
C07845=1074.209,323.205,405.359,175.017,29.765,155.296
C07846=1074.202,322.957,405.391,175.013,29.760,155.295
C07847=1074.196,322.709,405.424,175.011,29.756,155.294
C07848=1074.190,322.462,405.457,175.007,29.751,155.293
C07849=1074.184,322.213,405.491,175.004,29.746,155.293
C07850=1074.178,321.965,405.524,175.001,29.742,155.292
C07851=1074.172,321.718,405.557,174.998,29.737,155.291
C07852=1074.166,321.470,405.591,174.994,29.732,155.290
C07853=1074.160,321.223,405.623,174.992,29.728,155.289
C07854=1074.153,320.975,405.656,174.988,29.723,155.289
C07855=1074.148,320.727,405.689,174.986,29.719,155.288
C07856=1074.141,320.480,405.722,174.982,29.714,155.287
C07857=1074.136,320.232,405.756,174.979,29.709,155.286
C07858=1074.130,319.984,405.788,174.976,29.705,155.285
C07859=1074.124,319.736,405.822,174.973,29.700,155.285
C07860=1074.118,319.488,405.854,174.970,29.696,155.284
C07861=1074.112,319.241,405.886,174.967,29.691,155.283
C07862=1074.106,318.993,405.920,174.964,29.686,155.282
C07863=1074.100,318.745,405.953,174.961,29.682,155.281
C07864=1074.094,318.497,405.985,174.958,29.677,155.281
C07865=1074.088,318.250,406.019,174.955,29.673,155.280
C07866=1074.083,318.030,406.047,174.952,29.668,155.279
C07867=1074.078,317.809,406.077,174.949,29.664,155.278
C07868=1074.072,317.589,406.106,174.946,29.660,155.278
C07869=1074.067,317.369,406.135,174.944,29.656,155.277
C07870=1074.062,317.149,406.165,174.941,29.652,155.276
C07871=1074.057,316.929,406.194,174.939,29.648,155.275
C07872=1074.051,316.708,406.223,174.935,29.644,155.275
C07873=1074.046,316.488,406.251,174.933,29.640,155.274
C07874=1074.040,316.240,406.284,174.930,29.636,155.273
C07875=1074.034,315.993,406.317,174.927,29.630,155.272
C07876=1074.028,315.745,406.349,174.924,29.626,155.272
C07877=1074.022,315.497,406.382,174.921,29.622,155.271
C07878=1074.016,315.249,406.415,174.918,29.617,155.270
C07879=1074.011,315.002,406.447,174.915,29.613,155.269
C07880=1074.005,314.754,406.480,174.912,29.608,155.269
C07881=1073.999,314.506,406.513,174.909,29.604,155.268
C07882=1073.993,314.258,406.545,174.906,29.599,155.267
C07883=1073.987,314.010,406.578,174.903,29.595,155.266
C07884=1073.981,313.762,406.610,174.900,29.590,155.265
C07885=1073.974,313.514,406.642,174.897,29.586,155.265
C07886=1073.968,313.266,406.674,174.894,29.581,155.264
C07887=1073.961,313.019,406.706,174.890,29.577,155.263
C07888=1073.955,312.771,406.738,174.888,29.573,155.262
C07889=1073.949,312.523,406.771,174.884,29.568,155.262
C07890=1073.943,312.275,406.803,174.882,29.564,155.261
C07891=1073.937,312.028,406.836,174.878,29.560,155.260
C07892=1073.931,311.780,406.868,174.876,29.555,155.259
C07893=1073.925,311.532,406.900,174.872,29.551,155.259
C07894=1073.918,311.284,406.932,174.870,29.546,155.258
C07895=1073.912,311.036,406.964,174.866,29.542,155.257
C07896=1073.906,310.789,406.997,174.864,29.538,155.256
C07897=1073.901,310.541,407.028,174.861,29.533,155.256
C07898=1073.895,310.293,407.060,174.858,29.529,155.255
C07899=1073.888,310.045,407.092,174.855,29.525,155.254
C07900=1073.882,309.797,407.124,174.851,29.520,155.253
C07901=1073.876,309.549,407.156,174.849,29.516,155.253
C07902=1073.870,309.301,407.189,174.845,29.511,155.252
C07903=1073.864,309.054,407.221,174.843,29.507,155.251
C07904=1073.857,308.806,407.252,174.839,29.503,155.251
C07905=1073.851,308.558,407.284,174.837,29.498,155.250
C07906=1073.845,308.310,407.316,174.833,29.494,155.249
C07907=1073.840,308.062,407.348,174.831,29.490,155.248
C07908=1073.834,307.815,407.381,174.827,29.485,155.248
C07909=1073.827,307.567,407.412,174.825,29.481,155.247
C07910=1073.822,307.319,407.444,174.821,29.477,155.246
C07911=1073.816,307.071,407.476,174.819,29.472,155.245
C07912=1073.810,306.823,407.508,174.815,29.468,155.245
C07913=1073.803,306.576,407.539,174.813,29.464,155.244
C07914=1073.797,306.327,407.571,174.810,29.459,155.243
C07915=1073.791,306.079,407.603,174.807,29.455,155.242
C07916=1073.786,305.832,407.635,174.804,29.451,155.242
C07917=1073.779,305.584,407.667,174.801,29.446,155.241
C07918=1073.773,305.336,407.699,174.799,29.442,155.240
C07919=1073.768,305.089,407.731,174.795,29.438,155.240
C07920=1073.761,304.841,407.762,174.793,29.433,155.239
C07921=1073.755,304.592,407.794,174.789,29.429,155.238
C07922=1073.751,304.374,407.821,174.787,29.425,155.237
C07923=1073.746,304.155,407.849,174.784,29.421,155.237
C07924=1073.740,303.937,407.877,174.782,29.418,155.236
C07925=1073.735,303.718,407.905,174.779,29.414,155.235
C07926=1073.729,303.500,407.933,174.777,29.410,155.235
C07927=1073.724,303.281,407.961,174.774,29.406,155.234
C07928=1073.719,303.063,407.989,174.772,29.402,155.233
C07929=1073.714,302.844,408.017,174.769,29.398,155.233
C07930=1073.708,302.597,408.048,174.766,29.394,155.232
C07931=1073.701,302.349,408.080,174.763,29.390,155.231
C07932=1073.696,302.101,408.112,174.760,29.385,155.231
C07933=1073.690,301.852,408.143,174.757,29.381,155.230
C07934=1073.684,301.605,408.174,174.755,29.377,155.229
C07935=1073.678,301.357,408.206,174.751,29.373,155.229
C07936=1073.672,301.110,408.237,174.749,29.368,155.228
C07937=1073.666,300.861,408.269,174.745,29.364,155.227
C07938=1073.661,300.613,408.300,174.743,29.360,155.226
C07939=1073.654,300.365,408.331,174.739,29.355,155.226
C07940=1073.649,300.118,408.363,174.737,29.351,155.225
C07941=1073.643,299.869,408.394,174.734,29.347,155.224
C07942=1073.637,299.622,408.426,174.731,29.342,155.223
C07943=1073.631,299.374,408.458,174.729,29.339,155.223
C07944=1073.626,299.126,408.488,174.725,29.334,155.222
C07945=1073.620,298.878,408.520,174.723,29.329,155.221
C07946=1073.614,298.630,408.552,174.720,29.326,155.220
C07947=1073.608,298.382,408.582,174.717,29.321,155.220
C07948=1073.602,298.134,408.614,174.714,29.317,155.219
C07949=1073.596,297.886,408.644,174.711,29.312,155.218
C07950=1073.591,297.639,408.676,174.708,29.308,155.218
C07951=1073.585,297.390,408.707,174.706,29.304,155.217
C07952=1073.579,297.143,408.738,174.702,29.299,155.216
C07953=1073.573,296.894,408.769,174.700,29.296,155.215
C07954=1073.567,296.647,408.801,174.697,29.291,155.215
C07955=1073.561,296.398,408.831,174.694,29.287,155.214
C07956=1073.555,296.151,408.862,174.692,29.283,155.213
C07957=1073.549,295.902,408.894,174.688,29.279,155.213
C07958=1073.543,295.654,408.924,174.686,29.275,155.212
C07959=1073.537,295.407,408.955,174.683,29.271,155.211
C07960=1073.532,295.158,408.987,174.680,29.266,155.211
C07961=1073.525,294.911,409.018,174.677,29.262,155.210
C07962=1073.519,294.663,409.048,174.674,29.258,155.209
C07963=1073.513,294.415,409.079,174.671,29.254,155.208
C07964=1073.508,294.167,409.110,174.669,29.250,155.208
C07965=1073.501,293.919,409.141,174.665,29.245,155.207
C07966=1073.496,293.671,409.171,174.663,29.241,155.206
C07967=1073.489,293.422,409.202,174.660,29.237,155.206
C07968=1073.483,293.175,409.233,174.657,29.233,155.205
C07969=1073.478,292.927,409.264,174.655,29.229,155.204
C07970=1073.472,292.678,409.295,174.652,29.225,155.204
C07971=1073.466,292.431,409.325,174.649,29.220,155.203
C07972=1073.460,292.183,409.356,174.646,29.216,155.202
C07973=1073.453,291.935,409.387,174.644,29.212,155.202
C07974=1073.448,291.687,409.418,174.640,29.208,155.201
C07975=1073.442,291.439,409.448,174.638,29.204,155.200
C07976=1073.436,291.190,409.479,174.635,29.200,155.200
C07977=1073.430,290.943,409.509,174.632,29.196,155.199
C07978=1073.424,290.732,409.535,174.629,29.192,155.198
C07979=1073.420,290.520,409.562,174.628,29.189,155.198
C07980=1073.414,290.309,409.587,174.625,29.185,155.197
C07981=1073.410,290.098,409.614,174.623,29.182,155.196
C07982=1073.404,289.886,409.639,174.620,29.178,155.196
C07983=1073.400,289.676,409.666,174.618,29.174,155.195
C07984=1073.395,289.465,409.692,174.615,29.171,155.195
C07985=1073.390,289.253,409.718,174.614,29.168,155.194
C07986=1073.384,289.005,409.748,174.610,29.163,155.193
C07987=1073.378,288.756,409.779,174.608,29.159,155.193
C07988=1073.372,288.509,409.809,174.605,29.155,155.192
C07989=1073.366,288.261,409.839,174.602,29.151,155.191
C07990=1073.359,288.013,409.870,174.599,29.147,155.191
C07991=1073.353,287.765,409.900,174.597,29.143,155.190
C07992=1073.347,287.517,409.930,174.593,29.139,155.189
C07993=1073.342,287.269,409.961,174.591,29.135,155.189
C07994=1073.335,287.021,409.991,174.588,29.131,155.188
C07995=1073.330,286.772,410.021,174.585,29.127,155.187
C07996=1073.324,286.524,410.051,174.583,29.123,155.187
C07997=1073.318,286.277,410.082,174.580,29.118,155.186
C07998=1073.312,286.028,410.112,174.578,29.114,155.185
C07999=1073.306,285.780,410.143,174.574,29.110,155.185
C08000=1073.300,285.532,410.173,174.572,29.106,155.184
C08001=1073.295,285.284,410.203,174.569,29.103,155.183
C08002=1073.289,285.036,410.233,174.566,29.098,155.183
C08003=1073.282,284.788,410.263,174.563,29.094,155.182
C08004=1073.276,284.540,410.294,174.561,29.090,155.181
C08005=1073.270,284.292,410.323,174.558,29.086,155.181
C08006=1073.264,284.044,410.354,174.555,29.082,155.180
C08007=1073.259,283.796,410.384,174.553,29.078,155.179
C08008=1073.253,283.548,410.414,174.550,29.074,155.179
C08009=1073.247,283.299,410.444,174.548,29.070,155.178
C08010=1073.241,283.051,410.475,174.544,29.066,155.177
C08011=1073.235,282.803,410.504,174.542,29.062,155.177
C08012=1073.229,282.555,410.534,174.539,29.058,155.176
C08013=1073.223,282.307,410.564,174.536,29.054,155.175
C08014=1073.217,282.059,410.594,174.533,29.049,155.175
C08015=1073.212,281.811,410.624,174.531,29.045,155.174
C08016=1073.206,281.563,410.654,174.529,29.041,155.173
C08017=1073.200,281.315,410.684,174.525,29.037,155.173
C08018=1073.194,281.067,410.713,174.523,29.033,155.172
C08019=1073.188,280.818,410.744,174.520,29.029,155.171
C08020=1073.182,280.570,410.774,174.518,29.025,155.171
C08021=1073.176,280.322,410.804,174.515,29.021,155.170
C08022=1073.170,280.074,410.833,174.512,29.017,155.169
C08023=1073.165,279.825,410.863,174.509,29.013,155.169
C08024=1073.159,279.578,410.893,174.507,29.009,155.168
C08025=1073.152,279.329,410.922,174.504,29.005,155.167
C08026=1073.147,279.082,410.952,174.501,29.001,155.167
C08027=1073.140,278.834,410.982,174.499,28.997,155.166
C08028=1073.135,278.585,411.011,174.496,28.993,155.165
C08029=1073.129,278.337,411.042,174.494,28.989,155.165
C08030=1073.123,278.089,411.071,174.490,28.985,155.164
C08031=1073.117,277.841,411.100,174.488,28.981,155.164
C08032=1073.112,277.593,411.131,174.485,28.977,155.163
C08033=1073.105,277.345,411.160,174.483,28.973,155.162
C08034=1073.095,276.932,411.209,174.478,28.966,155.161
C08035=1073.086,276.520,411.258,174.474,28.959,155.160
C08036=1073.076,276.107,411.307,174.470,28.953,155.159
C08037=1073.066,275.695,411.357,174.465,28.946,155.158
C08038=1073.060,275.447,411.386,174.462,28.942,155.157
C08039=1073.054,275.199,411.415,174.460,28.938,155.156
C08040=1073.048,274.950,411.444,174.457,28.934,155.156
C08041=1073.042,274.702,411.474,174.455,28.930,155.155
C08042=1073.036,274.454,411.503,174.451,28.926,155.155
C08043=1073.031,274.205,411.533,174.449,28.922,155.154
C08044=1073.024,273.958,411.562,174.446,28.918,155.153
C08045=1073.019,273.709,411.592,174.444,28.914,155.153
C08046=1073.013,273.462,411.621,174.442,28.910,155.152
C08047=1073.007,273.214,411.650,174.439,28.906,155.151
C08048=1073.001,272.965,411.679,174.436,28.902,155.151
C08049=1072.996,272.717,411.709,174.433,28.898,155.150
C08050=1072.989,272.469,411.738,174.431,28.894,155.149
C08051=1072.983,272.221,411.767,174.428,28.890,155.149
C08052=1072.978,271.972,411.797,174.426,28.886,155.148
C08053=1072.971,271.724,411.826,174.422,28.882,155.147
C08054=1072.966,271.476,411.855,174.420,28.878,155.147
C08055=1072.960,271.228,411.885,174.418,28.874,155.146
C08056=1072.953,270.979,411.914,174.415,28.870,155.145
C08057=1072.948,270.730,411.942,174.413,28.866,155.145
C08058=1072.942,270.482,411.972,174.410,28.862,155.144
C08059=1072.936,270.235,412.000,174.407,28.858,155.144
C08060=1072.931,269.986,412.030,174.404,28.854,155.143
C08061=1072.924,269.738,412.059,174.402,28.850,155.142
C08062=1072.918,269.490,412.088,174.400,28.846,155.142
C08063=1072.913,269.242,412.118,174.397,28.842,155.141
C08064=1072.907,268.993,412.146,174.395,28.839,155.140
C08065=1072.901,268.745,412.175,174.392,28.835,155.140
C08066=1072.895,268.497,412.204,174.389,28.831,155.139
C08067=1072.889,268.249,412.233,174.386,28.827,155.138
C08068=1072.883,268.000,412.262,174.384,28.823,155.138
C08069=1072.877,267.752,412.291,174.381,28.819,155.137
C08070=1072.871,267.504,412.320,174.379,28.815,155.137
C08071=1072.865,267.256,412.349,174.377,28.811,155.136
C08072=1072.860,267.007,412.377,174.374,28.807,155.135
C08073=1072.854,266.759,412.406,174.371,28.803,155.135
C08074=1072.848,266.511,412.435,174.368,28.799,155.134
C08075=1072.842,266.262,412.464,174.366,28.795,155.133
C08076=1072.835,266.014,412.493,174.363,28.791,155.133
C08077=1072.831,265.766,412.521,174.361,28.787,155.132
C08078=1072.825,265.518,412.550,174.359,28.783,155.131
C08079=1072.818,265.270,412.579,174.356,28.779,155.131
C08080=1072.812,265.021,412.608,174.354,28.776,155.130
C08081=1072.807,264.773,412.636,174.350,28.772,155.130
C08082=1072.801,264.525,412.665,174.348,28.768,155.129
C08083=1072.795,264.277,412.694,174.345,28.764,155.128
C08084=1072.789,264.027,412.723,174.343,28.760,155.128
C08085=1072.784,263.780,412.751,174.340,28.756,155.127
C08086=1072.773,263.371,412.798,174.336,28.749,155.126
C08087=1072.763,262.962,412.845,174.332,28.743,155.125
C08088=1072.754,262.553,412.892,174.328,28.737,155.124
C08089=1072.743,262.143,412.939,174.324,28.731,155.123
C08090=1072.737,261.895,412.967,174.321,28.726,155.122
C08091=1072.731,261.648,412.996,174.318,28.722,155.122
C08092=1072.725,261.399,413.024,174.316,28.718,155.121
C08093=1072.719,261.150,413.052,174.313,28.715,155.120
C08094=1072.713,260.902,413.082,174.311,28.711,155.120
C08095=1072.708,260.654,413.109,174.309,28.707,155.119
C08096=1072.702,260.405,413.138,174.306,28.703,155.119
C08097=1072.695,260.157,413.166,174.304,28.699,155.118
C08098=1072.689,259.909,413.194,174.301,28.696,155.117
C08099=1072.683,259.660,413.223,174.299,28.692,155.117
C08100=1072.677,259.412,413.251,174.296,28.688,155.116
C08101=1072.671,259.164,413.280,174.293,28.684,155.115
C08102=1072.665,258.916,413.307,174.291,28.680,155.115
C08103=1072.659,258.667,413.336,174.288,28.676,155.114
C08104=1072.653,258.418,413.364,174.286,28.672,155.114
C08105=1072.648,258.170,413.392,174.283,28.668,155.113
C08106=1072.642,257.922,413.421,174.281,28.664,155.112
C08107=1072.636,257.673,413.449,174.278,28.660,155.112
C08108=1072.630,257.426,413.477,174.276,28.656,155.111
C08109=1072.624,257.177,413.505,174.274,28.653,155.110
C08110=1072.618,256.929,413.533,174.271,28.649,155.110
C08111=1072.612,256.680,413.561,174.269,28.645,155.109
C08112=1072.606,256.432,413.589,174.266,28.641,155.109
C08113=1072.600,256.184,413.617,174.264,28.637,155.108
C08114=1072.594,255.935,413.645,174.261,28.633,155.107
C08115=1072.589,255.687,413.673,174.259,28.630,155.107
C08116=1072.582,255.438,413.701,174.257,28.626,155.106
C08117=1072.576,255.190,413.729,174.254,28.622,155.105
C08118=1072.571,254.942,413.758,174.251,28.617,155.105
C08119=1072.565,254.693,413.786,174.248,28.613,155.104
C08120=1072.559,254.445,413.813,174.246,28.609,155.104
C08121=1072.553,254.196,413.841,174.244,28.605,155.103
C08122=1072.548,253.948,413.869,174.241,28.602,155.102
C08123=1072.542,253.700,413.897,174.239,28.598,155.102
C08124=1072.536,253.452,413.925,174.236,28.594,155.101
C08125=1072.530,253.203,413.953,174.234,28.590,155.100
C08126=1072.525,252.955,413.981,174.231,28.586,155.100
C08127=1072.519,252.706,414.009,174.229,28.582,155.099
C08128=1072.513,252.458,414.037,174.227,28.578,155.098
C08129=1072.507,252.210,414.065,174.224,28.574,155.098
C08130=1072.501,251.962,414.093,174.222,28.570,155.097
C08131=1072.495,251.713,414.120,174.219,28.567,155.097
C08132=1072.490,251.465,414.148,174.217,28.563,155.096
C08133=1072.484,251.216,414.176,174.214,28.559,155.095
C08134=1072.477,250.968,414.204,174.212,28.555,155.095
C08135=1072.472,250.719,414.232,174.210,28.551,155.094
C08136=1072.467,250.471,414.259,174.207,28.547,155.093
C08137=1072.461,250.222,414.288,174.205,28.543,155.093
C08138=1072.451,249.811,414.334,174.201,28.536,155.092
C08139=1072.441,249.399,414.379,174.197,28.530,155.091
C08140=1072.432,248.988,414.425,174.193,28.523,155.090
C08141=1072.422,248.576,414.470,174.189,28.517,155.089
C08142=1072.416,248.328,414.499,174.186,28.513,155.088
C08143=1072.411,248.080,414.527,174.184,28.509,155.087
C08144=1072.405,247.831,414.554,174.182,28.505,155.087
C08145=1072.399,247.583,414.582,174.179,28.501,155.086
C08146=1072.394,247.335,414.610,174.177,28.497,155.085
C08147=1072.388,247.085,414.637,174.174,28.493,155.085
C08148=1072.382,246.837,414.665,174.172,28.489,155.084
C08149=1072.377,246.589,414.691,174.171,28.485,155.083
C08150=1072.371,246.340,414.720,174.168,28.481,155.083
C08151=1072.365,246.092,414.746,174.166,28.478,155.082
C08152=1072.359,245.843,414.775,174.163,28.474,155.082
C08153=1072.353,245.595,414.801,174.161,28.470,155.081
C08154=1072.347,245.347,414.829,174.159,28.466,155.080
C08155=1072.341,245.098,414.856,174.156,28.462,155.080
C08156=1072.335,244.850,414.884,174.154,28.458,155.079
C08157=1072.330,244.601,414.911,174.151,28.454,155.078
C08158=1072.324,244.353,414.938,174.149,28.450,155.078
C08159=1072.318,244.104,414.965,174.147,28.446,155.077
C08160=1072.312,243.856,414.993,174.144,28.442,155.077
C08161=1072.306,243.607,415.020,174.142,28.438,155.076
C08162=1072.301,243.359,415.047,174.139,28.434,155.075
C08163=1072.295,243.111,415.075,174.137,28.430,155.075
C08164=1072.289,242.862,415.102,174.135,28.426,155.074
C08165=1072.284,242.613,415.129,174.132,28.422,155.073
C08166=1072.278,242.366,415.156,174.130,28.419,155.073
C08167=1072.271,242.116,415.183,174.127,28.415,155.072
C08168=1072.265,241.868,415.210,174.125,28.411,155.072
C08169=1072.260,241.620,415.238,174.123,28.407,155.071
C08170=1072.254,241.371,415.265,174.120,28.403,155.070
C08171=1072.248,241.123,415.292,174.119,28.400,155.070
C08172=1072.242,240.874,415.318,174.116,28.396,155.069
C08173=1072.236,240.627,415.346,174.114,28.392,155.068
C08174=1072.230,240.377,415.373,174.112,28.388,155.068
C08175=1072.225,240.129,415.400,174.109,28.383,155.067
C08176=1072.219,239.880,415.427,174.107,28.380,155.067
C08177=1072.212,239.631,415.454,174.104,28.376,155.066
C08178=1072.206,239.384,415.481,174.102,28.372,155.065
C08179=1072.201,239.135,415.508,174.100,28.368,155.065
C08180=1072.196,238.887,415.535,174.097,28.364,155.064
C08181=1072.189,238.638,415.562,174.095,28.361,155.064
C08182=1072.183,238.389,415.588,174.092,28.357,155.063
C08183=1072.178,238.141,415.615,174.090,28.353,155.062
C08184=1072.172,237.892,415.642,174.088,28.349,155.062
C08185=1072.165,237.643,415.669,174.086,28.345,155.061
C08186=1072.159,237.396,415.696,174.084,28.341,155.060
C08187=1072.154,237.147,415.723,174.081,28.337,155.060
C08188=1072.149,236.899,415.750,174.079,28.333,155.059
C08189=1072.142,236.650,415.777,174.077,28.329,155.059
C08190=1072.133,236.232,415.821,174.073,28.323,155.057
C08191=1072.123,235.814,415.866,174.069,28.316,155.056
C08192=1072.113,235.396,415.911,174.065,28.309,155.055
C08193=1072.104,234.978,415.956,174.061,28.303,155.054
C08194=1072.098,234.729,415.983,174.059,28.299,155.054
C08195=1072.091,234.480,416.010,174.057,28.295,155.053
C08196=1072.086,234.232,416.037,174.055,28.291,155.052
C08197=1072.080,233.983,416.063,174.052,28.287,155.052
C08198=1072.074,233.735,416.090,174.050,28.283,155.051
C08199=1072.068,233.487,416.117,174.048,28.279,155.051
C08200=1072.063,233.238,416.143,174.045,28.275,155.050
C08201=1072.057,232.989,416.169,174.043,28.272,155.049
C08202=1072.051,232.741,416.196,174.041,28.268,155.049
C08203=1072.045,232.492,416.223,174.039,28.264,155.048
C08204=1072.039,232.244,416.250,174.037,28.260,155.047
C08205=1072.034,231.995,416.275,174.034,28.256,155.047
C08206=1072.028,231.746,416.302,174.032,28.252,155.046
C08207=1072.022,231.498,416.329,174.029,28.248,155.046
C08208=1072.016,231.250,416.355,174.027,28.244,155.045
C08209=1072.010,231.001,416.381,174.025,28.240,155.044
C08210=1072.004,230.752,416.407,174.023,28.236,155.044
C08211=1071.999,230.504,416.434,174.021,28.232,155.043
C08212=1071.993,230.256,416.461,174.019,28.228,155.042
C08213=1071.987,230.007,416.487,174.016,28.224,155.042
C08214=1071.982,229.788,416.510,174.015,28.221,155.041
C08215=1071.977,229.569,416.533,174.012,28.218,155.041
C08216=1071.972,229.351,416.556,174.011,28.214,155.040
C08217=1071.966,229.131,416.580,174.008,28.211,155.040
C08218=1071.961,228.913,416.603,174.007,28.208,155.039
C08219=1071.956,228.694,416.626,174.004,28.204,155.039
C08220=1071.951,228.475,416.648,174.002,28.201,155.038
C08221=1071.945,228.256,416.672,174.001,28.197,155.037
C08222=1071.939,228.008,416.698,173.998,28.194,155.037
C08223=1071.933,227.759,416.724,173.996,28.190,155.036
C08224=1071.928,227.511,416.751,173.994,28.185,155.036
C08225=1071.922,227.262,416.777,173.992,28.182,155.035
C08226=1071.916,227.014,416.803,173.990,28.178,155.034
C08227=1071.910,226.765,416.829,173.987,28.174,155.034
C08228=1071.905,226.516,416.855,173.985,28.170,155.033
C08229=1071.898,226.268,416.881,173.983,28.166,155.033
C08230=1071.893,226.019,416.907,173.980,28.162,155.032
C08231=1071.887,225.771,416.934,173.979,28.158,155.031
C08232=1071.881,225.522,416.959,173.977,28.154,155.031
C08233=1071.875,225.273,416.985,173.974,28.150,155.030
C08234=1071.869,225.025,417.012,173.972,28.147,155.029
C08235=1071.863,224.776,417.037,173.969,28.143,155.029
C08236=1071.857,224.528,417.064,173.968,28.139,155.028
C08237=1071.852,224.279,417.090,173.966,28.135,155.027
C08238=1071.845,224.031,417.116,173.963,28.131,155.027
C08239=1071.840,223.782,417.142,173.961,28.127,155.026
C08240=1071.834,223.533,417.168,173.959,28.123,155.026
C08241=1071.828,223.285,417.194,173.957,28.119,155.025
C08242=1071.823,223.042,417.219,173.955,28.115,155.024
C08243=1071.818,222.798,417.244,173.952,28.111,155.024
C08244=1071.812,222.556,417.269,173.950,28.107,155.023
C08245=1071.806,222.313,417.295,173.949,28.104,155.022
C08246=1071.800,222.070,417.320,173.946,28.100,155.022
C08247=1071.795,221.827,417.345,173.944,28.096,155.021
C08248=1071.789,221.584,417.371,173.942,28.092,155.021
C08249=1071.783,221.341,417.396,173.940,28.088,155.020
C08250=1071.778,221.093,417.422,173.938,28.084,155.019
C08251=1071.772,220.844,417.447,173.935,28.081,155.019
C08252=1071.765,220.595,417.472,173.933,28.077,155.018
C08253=1071.760,220.346,417.498,173.931,28.073,155.018
C08254=1071.754,220.098,417.524,173.929,28.069,155.017
C08255=1071.748,219.849,417.550,173.927,28.065,155.016
C08256=1071.742,219.601,417.576,173.925,28.061,155.016
C08257=1071.736,219.352,417.601,173.922,28.057,155.015
C08258=1071.730,219.103,417.627,173.921,28.053,155.014
C08259=1071.724,218.854,417.652,173.919,28.049,155.014
C08260=1071.719,218.606,417.678,173.916,28.045,155.013
C08261=1071.713,218.358,417.704,173.914,28.041,155.013
C08262=1071.706,218.109,417.729,173.912,28.037,155.012
C08263=1071.701,217.860,417.755,173.910,28.033,155.011
C08264=1071.695,217.612,417.781,173.908,28.029,155.011
C08265=1071.689,217.363,417.806,173.906,28.026,155.010
C08266=1071.683,217.114,417.832,173.903,28.022,155.009
C08267=1071.677,216.866,417.857,173.902,28.018,155.009
C08268=1071.672,216.617,417.883,173.899,28.014,155.008
C08269=1071.666,216.368,417.908,173.897,28.010,155.008
C08270=1071.660,216.120,417.933,173.895,28.006,155.007
C08271=1071.654,215.871,417.959,173.893,28.002,155.006
C08272=1071.648,215.623,417.984,173.891,27.998,155.006
C08273=1071.643,215.374,418.010,173.889,27.994,155.005
C08274=1071.637,215.125,418.036,173.886,27.990,155.004
C08275=1071.631,214.876,418.061,173.885,27.986,155.004
C08276=1071.626,214.628,418.086,173.883,27.982,155.003
C08277=1071.620,214.380,418.112,173.880,27.979,155.002
C08278=1071.613,214.131,418.137,173.878,27.975,155.002
C08279=1071.608,213.881,418.162,173.877,27.971,155.001
C08280=1071.603,213.633,418.187,173.874,27.967,155.001
C08281=1071.596,213.385,418.213,173.872,27.963,155.000
C08282=1071.590,213.136,418.238,173.870,27.959,154.999
C08283=1071.585,212.887,418.264,173.868,27.955,154.999
C08284=1071.579,212.639,418.289,173.866,27.951,154.998
C08285=1071.573,212.390,418.314,173.864,27.947,154.997
C08286=1071.567,212.141,418.339,173.861,27.943,154.997
C08287=1071.561,211.892,418.364,173.860,27.939,154.996
C08288=1071.556,211.644,418.390,173.858,27.935,154.995
C08289=1071.550,211.395,418.415,173.855,27.931,154.995
C08290=1071.544,211.146,418.440,173.853,27.927,154.994
C08291=1071.538,210.898,418.465,173.852,27.923,154.993
C08292=1071.532,210.650,418.490,173.849,27.919,154.993
C08293=1071.526,210.401,418.515,173.847,27.915,154.992
C08294=1071.521,210.151,418.541,173.846,27.911,154.992
C08295=1071.515,209.903,418.566,173.843,27.907,154.991
C08296=1071.509,209.655,418.591,173.841,27.903,154.990
C08297=1071.503,209.405,418.616,173.839,27.899,154.990
C08298=1071.498,209.196,418.637,173.837,27.896,154.989
C08299=1071.493,208.984,418.658,173.836,27.893,154.989
C08300=1071.489,208.773,418.679,173.834,27.889,154.988
C08301=1071.483,208.562,418.701,173.832,27.886,154.988
C08302=1071.478,208.351,418.722,173.830,27.883,154.987
C08303=1071.473,208.140,418.742,173.829,27.879,154.987
C08304=1071.468,207.929,418.764,173.827,27.876,154.986
C08305=1071.439,206.676,418.887,173.692,27.803,154.983
C08306=1071.434,206.428,418.911,173.690,27.801,154.983
C08307=1071.428,206.178,418.936,173.688,27.798,154.983
C08308=1071.422,205.930,418.959,173.685,27.795,154.982
C08309=1071.417,205.681,418.983,173.683,27.791,154.982
C08310=1071.411,205.432,419.008,173.681,27.788,154.981
C08311=1071.406,205.183,419.032,173.679,27.785,154.981
C08312=1071.400,204.935,419.056,173.676,27.782,154.981
C08313=1071.394,204.686,419.081,173.674,27.779,154.980
C08314=1071.388,204.437,419.105,173.672,27.776,154.980
C08315=1071.383,204.189,419.129,173.670,27.773,154.979
C08316=1071.376,203.940,419.153,173.667,27.770,154.979
C08317=1071.371,203.691,419.177,173.665,27.767,154.978
C08318=1071.366,203.443,419.202,173.663,27.764,154.978
C08319=1071.360,203.194,419.225,173.661,27.761,154.978
C08320=1071.354,202.944,419.249,173.659,27.758,154.977
C08321=1071.349,202.696,419.273,173.657,27.755,154.977
C08322=1071.344,202.447,419.298,173.655,27.752,154.976
C08323=1071.337,202.198,419.322,173.652,27.749,154.976
C08324=1071.332,201.950,419.346,173.650,27.746,154.976
C08325=1071.326,201.701,419.370,173.648,27.743,154.975
C08326=1071.320,201.451,419.394,173.646,27.740,154.975
C08327=1071.314,201.203,419.417,173.643,27.737,154.974
C08328=1071.309,200.955,419.442,173.641,27.734,154.974
C08329=1071.303,200.706,419.465,173.639,27.732,154.974
C08330=1071.296,200.457,419.488,173.637,27.729,154.973
C08331=1071.291,200.208,419.513,173.634,27.726,154.973
C08332=1071.285,199.960,419.536,173.633,27.723,154.972
C08333=1071.279,199.711,419.561,173.630,27.719,154.972
C08334=1071.273,199.462,419.584,173.628,27.716,154.972
C08335=1071.268,199.213,419.608,173.626,27.714,154.971
C08336=1071.262,198.965,419.632,173.624,27.711,154.971
C08337=1071.256,198.715,419.656,173.621,27.708,154.970
C08338=1071.250,198.467,419.679,173.619,27.705,154.970
C08339=1071.244,198.218,419.703,173.617,27.702,154.970
C08340=1071.239,197.969,419.727,173.615,27.699,154.969
C08341=1071.233,197.720,419.751,173.612,27.696,154.969
C08342=1071.228,197.471,419.774,173.611,27.693,154.968
C08343=1071.222,197.223,419.798,173.608,27.690,154.968
C08344=1071.216,196.974,419.822,173.606,27.687,154.968
C08345=1071.211,196.725,419.845,173.604,27.684,154.967
C08346=1071.204,196.476,419.869,173.602,27.681,154.967
C08347=1071.199,196.227,419.893,173.600,27.678,154.966
C08348=1071.193,195.979,419.916,173.598,27.676,154.966
C08349=1071.188,195.730,419.940,173.596,27.673,154.966
C08350=1071.182,195.481,419.964,173.593,27.670,154.965
C08351=1071.176,195.232,419.987,173.592,27.667,154.965
C08352=1071.170,194.983,420.011,173.589,27.664,154.964
C08353=1071.165,194.734,420.034,173.587,27.661,154.964
C08354=1071.159,194.486,420.058,173.585,27.658,154.964
C08355=1071.154,194.237,420.081,173.583,27.655,154.963
C08356=1071.148,193.988,420.105,173.580,27.652,154.963
C08357=1071.143,193.739,420.128,173.579,27.649,154.962
C08358=1071.136,193.490,420.152,173.576,27.646,154.962
C08359=1071.130,193.241,420.175,173.574,27.643,154.962
C08360=1071.125,192.993,420.200,173.572,27.641,154.961
C08361=1071.119,192.744,420.223,173.570,27.638,154.961
C08362=1071.113,192.495,420.246,173.567,27.635,154.960
C08363=1071.108,192.246,420.270,173.566,27.632,154.960
C08364=1071.102,191.997,420.293,173.563,27.629,154.960
C08365=1071.097,191.749,420.316,173.562,27.626,154.959
C08366=1071.090,191.467,420.343,173.559,27.623,154.959
C08367=1071.084,191.186,420.369,173.557,27.619,154.958
C08368=1071.078,190.903,420.397,173.555,27.616,154.958
C08369=1071.071,190.621,420.423,173.552,27.613,154.957
C08370=1071.066,190.372,420.446,173.550,27.610,154.957
C08371=1071.060,190.124,420.469,173.547,27.607,154.957
C08372=1071.054,189.875,420.492,173.546,27.604,154.956
C08373=1071.049,189.626,420.516,173.543,27.601,154.956
C08374=1071.043,189.377,420.539,173.542,27.598,154.955
C08375=1071.037,189.129,420.563,173.539,27.595,154.955
C08376=1071.032,188.879,420.586,173.537,27.592,154.955
C08377=1071.026,188.631,420.609,173.535,27.589,154.954
C08378=1071.021,188.382,420.632,173.533,27.586,154.954
C08379=1071.016,188.132,420.656,173.531,27.583,154.953
C08380=1071.010,187.884,420.679,173.529,27.580,154.953
C08381=1071.004,187.635,420.702,173.527,27.577,154.953
C08382=1070.998,187.386,420.725,173.525,27.575,154.952
C08383=1070.993,187.137,420.749,173.523,27.572,154.952
C08384=1070.987,186.888,420.772,173.521,27.568,154.951
C08385=1070.982,186.639,420.795,173.519,27.565,154.951
C08386=1070.976,186.391,420.819,173.517,27.563,154.951
C08387=1070.971,186.142,420.842,173.515,27.560,154.950
C08388=1070.965,185.894,420.864,173.512,27.557,154.950
C08389=1070.960,185.645,420.887,173.511,27.554,154.949
C08390=1070.955,185.396,420.911,173.508,27.551,154.949
C08391=1070.949,185.147,420.934,173.507,27.548,154.949
C08392=1070.943,184.898,420.957,173.504,27.545,154.948
C08393=1070.938,184.649,420.980,173.502,27.542,154.948
C08394=1070.932,184.400,421.003,173.500,27.539,154.947
C08395=1070.926,184.151,421.026,173.498,27.537,154.947
C08396=1070.920,183.902,421.048,173.496,27.534,154.947
C08397=1070.915,183.653,421.071,173.494,27.531,154.946
C08398=1070.908,183.405,421.094,173.492,27.528,154.946
C08399=1070.902,183.156,421.117,173.490,27.525,154.946
C08400=1070.897,182.907,421.140,173.487,27.523,154.945
C08401=1070.891,182.658,421.163,173.486,27.520,154.945
C08402=1070.885,182.409,421.186,173.483,27.517,154.944
C08403=1070.879,182.160,421.209,173.482,27.514,154.944
C08404=1070.873,181.912,421.231,173.479,27.511,154.944
C08405=1070.867,181.663,421.254,173.478,27.509,154.943
C08406=1070.862,181.414,421.277,173.475,27.506,154.943
C08407=1070.856,181.165,421.300,173.474,27.503,154.943
C08408=1070.850,180.915,421.322,173.471,27.500,154.942
C08409=1070.844,180.667,421.344,173.469,27.497,154.942
C08410=1070.838,180.418,421.367,173.467,27.495,154.942
C08411=1070.832,180.169,421.390,173.465,27.492,154.941
C08412=1070.827,179.920,421.413,173.463,27.489,154.941
C08413=1070.821,179.671,421.436,173.461,27.486,154.940
C08414=1070.815,179.422,421.458,173.459,27.484,154.940
C08415=1070.809,179.173,421.481,173.457,27.481,154.940
C08416=1070.803,178.924,421.504,173.455,27.478,154.939
C08417=1070.798,178.675,421.527,173.453,27.475,154.939
C08418=1070.792,178.426,421.549,173.451,27.473,154.938
C08419=1070.786,178.177,421.571,173.449,27.469,154.938
C08420=1070.780,177.928,421.594,173.447,27.467,154.938
C08421=1070.774,177.679,421.617,173.445,27.464,154.937
C08422=1070.769,177.431,421.640,173.443,27.461,154.937
C08423=1070.763,177.182,421.661,173.441,27.458,154.937
C08424=1070.757,176.933,421.684,173.439,27.456,154.936
C08425=1070.752,176.684,421.707,173.437,27.453,154.936
C08426=1070.746,176.435,421.729,173.435,27.450,154.936
C08427=1070.740,176.186,421.752,173.433,27.447,154.935
C08428=1070.734,175.937,421.775,173.431,27.444,154.935
C08429=1070.729,175.688,421.797,173.429,27.442,154.934
C08430=1070.721,175.406,421.823,173.427,27.439,154.934
C08431=1070.715,175.124,421.848,173.424,27.435,154.933
C08432=1070.709,174.842,421.873,173.422,27.432,154.933
C08433=1070.703,174.559,421.899,173.420,27.429,154.933
C08434=1070.697,174.312,421.921,173.418,27.426,154.932
C08435=1070.691,174.062,421.943,173.416,27.423,154.932
C08436=1070.686,173.813,421.966,173.414,27.420,154.932
C08437=1070.680,173.564,421.988,173.412,27.418,154.931
C08438=1070.674,173.315,422.011,173.410,27.415,154.931
C08439=1070.669,173.067,422.033,173.408,27.412,154.930
C08440=1070.663,172.817,422.056,173.406,27.409,154.930
C08441=1070.657,172.569,422.078,173.404,27.407,154.930
C08442=1070.651,172.319,422.100,173.402,27.404,154.929
C08443=1070.646,172.070,422.123,173.401,27.401,154.929
C08444=1070.640,171.822,422.144,173.398,27.398,154.928
C08445=1070.634,171.573,422.167,173.397,27.396,154.928
C08446=1070.629,171.323,422.190,173.394,27.393,154.928
C08447=1070.622,171.075,422.212,173.393,27.390,154.927
C08448=1070.618,170.826,422.234,173.390,27.387,154.927
C08449=1070.612,170.577,422.257,173.389,27.384,154.927
C08450=1070.606,170.328,422.278,173.387,27.381,154.926
C08451=1070.601,170.079,422.300,173.385,27.378,154.926
C08452=1070.595,169.830,422.323,173.383,27.375,154.925
C08453=1070.589,169.581,422.345,173.381,27.373,154.925
C08454=1070.583,169.332,422.368,173.379,27.370,154.925
C08455=1070.578,169.083,422.390,173.377,27.367,154.924
C08456=1070.572,168.834,422.411,173.375,27.364,154.924
C08457=1070.567,168.585,422.434,173.373,27.361,154.924
C08458=1070.562,168.336,422.456,173.371,27.359,154.923
C08459=1070.555,168.088,422.478,173.370,27.356,154.923
C08460=1070.550,167.838,422.501,173.367,27.353,154.922
C08461=1070.545,167.589,422.523,173.366,27.351,154.922
C08462=1070.539,167.341,422.545,173.363,27.348,154.922
C08463=1070.533,167.091,422.567,173.362,27.345,154.921
C08464=1070.528,166.843,422.588,173.359,27.342,154.921
C08465=1070.522,166.593,422.611,173.358,27.339,154.920
C08466=1070.516,166.344,422.634,173.356,27.336,154.920
C08467=1070.511,166.096,422.655,173.354,27.333,154.920
C08468=1070.505,165.846,422.677,173.353,27.330,154.919
C08469=1070.500,165.598,422.700,173.350,27.327,154.919
C08470=1070.494,165.349,422.721,173.349,27.325,154.918
C08471=1070.489,165.099,422.743,173.346,27.322,154.918
C08472=1070.483,164.851,422.765,173.345,27.319,154.918
C08473=1070.478,164.601,422.787,173.343,27.317,154.917
C08474=1070.473,164.353,422.810,173.341,27.314,154.917
C08475=1070.466,164.104,422.831,173.339,27.311,154.917
C08476=1070.461,163.855,422.853,173.337,27.308,154.916
C08477=1070.455,163.606,422.875,173.335,27.305,154.916
C08478=1070.450,163.357,422.897,173.334,27.302,154.915
C08479=1070.444,163.109,422.919,173.331,27.299,154.915
C08480=1070.439,162.859,422.941,173.330,27.296,154.915
C08481=1070.434,162.610,422.963,173.327,27.293,154.914
C08482=1070.428,162.361,422.985,173.326,27.291,154.914
C08483=1070.423,162.112,423.007,173.324,27.288,154.913
C08484=1070.417,161.863,423.028,173.322,27.285,154.913
C08485=1070.412,161.614,423.050,173.320,27.283,154.913
C08486=1070.406,161.365,423.072,173.318,27.279,154.912
C08487=1070.400,161.116,423.094,173.317,27.277,154.912
C08488=1070.394,160.868,423.116,173.315,27.274,154.912
C08489=1070.388,160.618,423.137,173.313,27.271,154.911
C08490=1070.384,160.370,423.159,173.311,27.268,154.911
C08491=1070.377,160.120,423.181,173.309,27.266,154.910
C08492=1070.371,159.871,423.203,173.307,27.263,154.910
C08493=1070.366,159.623,423.224,173.306,27.260,154.910
C08494=1070.359,159.340,423.248,173.303,27.257,154.909
C08495=1070.353,159.057,423.273,173.301,27.254,154.909
C08496=1070.346,158.775,423.297,173.299,27.251,154.908
C08497=1070.340,158.493,423.322,173.297,27.248,154.908
C08498=1070.334,158.243,423.344,173.295,27.245,154.908
C08499=1070.329,157.994,423.366,173.293,27.242,154.907
C08500=1070.323,157.745,423.386,173.292,27.240,154.907
C08501=1070.317,157.496,423.408,173.289,27.236,154.907
C08502=1070.311,157.247,423.429,173.288,27.234,154.906
C08503=1070.306,156.998,423.451,173.286,27.231,154.906
C08504=1070.300,156.749,423.473,173.284,27.228,154.905
C08505=1070.294,156.500,423.494,173.282,27.226,154.905
C08506=1070.288,156.251,423.516,173.280,27.223,154.905
C08507=1070.283,156.003,423.537,173.278,27.220,154.904
C08508=1070.277,155.753,423.559,173.277,27.217,154.904
C08509=1070.272,155.504,423.580,173.274,27.215,154.904
C08510=1070.266,155.255,423.601,173.273,27.212,154.903
C08511=1070.260,155.006,423.623,173.271,27.209,154.903
C08512=1070.254,154.757,423.644,173.269,27.206,154.902
C08513=1070.249,154.509,423.666,173.267,27.204,154.902
C08514=1070.243,154.259,423.687,173.266,27.201,154.902
C08515=1070.237,154.009,423.709,173.263,27.198,154.901
C08516=1070.232,153.761,423.730,173.262,27.195,154.901
C08517=1070.226,153.512,423.751,173.260,27.193,154.901
C08518=1070.220,153.263,423.773,173.258,27.190,154.900
C08519=1070.215,153.014,423.793,173.256,27.187,154.900
C08520=1070.209,152.765,423.815,173.255,27.184,154.899
C08521=1070.203,152.516,423.836,173.252,27.182,154.899
C08522=1070.197,152.266,423.857,173.251,27.179,154.899
C08523=1070.192,152.018,423.879,173.249,27.176,154.898
C08524=1070.186,151.769,423.900,173.247,27.173,154.898
C08525=1070.180,151.520,423.921,173.246,27.170,154.898
C08526=1070.174,151.270,423.942,173.244,27.168,154.897
C08527=1070.169,151.022,423.964,173.242,27.165,154.897
C08528=1070.162,150.773,423.985,173.240,27.162,154.897
C08529=1070.157,150.524,424.006,173.239,27.160,154.896
C08530=1070.152,150.275,424.027,173.236,27.157,154.896
C08531=1070.146,150.025,424.048,173.235,27.154,154.895
C08532=1070.140,149.777,424.069,173.233,27.151,154.895
C08533=1070.134,149.528,424.091,173.231,27.148,154.895
C08534=1070.129,149.278,424.112,173.229,27.146,154.894
C08535=1070.123,149.030,424.133,173.228,27.143,154.894
C08536=1070.117,148.780,424.154,173.225,27.140,154.894
C08537=1070.112,148.532,424.175,173.224,27.138,154.893
C08538=1070.106,148.282,424.197,173.222,27.135,154.893
C08539=1070.100,148.033,424.217,173.220,27.132,154.893
C08540=1070.094,147.784,424.239,173.218,27.129,154.892
C08541=1070.089,147.535,424.259,173.217,27.127,154.892
C08542=1070.083,147.286,424.281,173.214,27.124,154.891
C08543=1070.077,147.037,424.302,173.213,27.121,154.891
C08544=1070.072,146.788,424.323,173.211,27.119,154.891
C08545=1070.065,146.539,424.343,173.210,27.116,154.890
C08546=1070.060,146.290,424.364,173.207,27.113,154.890
C08547=1070.054,146.041,424.385,173.206,27.111,154.890
C08548=1070.048,145.792,424.407,173.205,27.108,154.889
C08549=1070.043,145.543,424.427,173.202,27.105,154.889
C08550=1070.037,145.293,424.449,173.201,27.102,154.888
C08551=1070.031,145.045,424.469,173.199,27.100,154.888
C08552=1070.026,144.795,424.489,173.197,27.097,154.888
C08553=1070.020,144.546,424.511,173.195,27.094,154.887
C08554=1070.014,144.297,424.531,173.194,27.092,154.887
C08555=1070.009,144.049,424.553,173.192,27.089,154.887
C08556=1070.002,143.799,424.573,173.190,27.086,154.886
C08557=1069.997,143.550,424.594,173.188,27.083,154.886
C08558=1069.990,143.267,424.618,173.186,27.080,154.885
C08559=1069.984,142.984,424.641,173.184,27.077,154.885
C08560=1069.978,142.702,424.665,173.182,27.074,154.885
C08561=1069.971,142.419,424.688,173.181,27.071,154.884
C08562=1069.965,142.169,424.709,173.178,27.068,154.884
C08563=1069.959,141.921,424.730,173.177,27.065,154.883
C08564=1069.954,141.672,424.751,173.175,27.063,154.883
C08565=1069.949,141.423,424.771,173.174,27.060,154.883
C08566=1069.942,141.174,424.792,173.171,27.057,154.882
C08567=1069.937,140.925,424.813,173.170,27.054,154.882
C08568=1069.932,140.675,424.833,173.168,27.052,154.882
C08569=1069.925,140.426,424.855,173.167,27.049,154.881
C08570=1069.919,140.177,424.875,173.164,27.046,154.881
C08571=1069.914,139.928,424.896,173.163,27.044,154.881
C08572=1069.908,139.679,424.917,173.161,27.041,154.880
C08573=1069.902,139.430,424.937,173.159,27.038,154.880
C08574=1069.897,139.181,424.958,173.157,27.035,154.879
C08575=1069.891,138.932,424.978,173.156,27.033,154.879
C08576=1069.885,138.683,424.999,173.154,27.030,154.879
C08577=1069.880,138.433,425.019,173.152,27.027,154.878
C08578=1069.874,138.185,425.039,173.151,27.025,154.878
C08579=1069.868,137.936,425.060,173.149,27.022,154.878
C08580=1069.862,137.686,425.081,173.148,27.019,154.877
C08581=1069.856,137.437,425.101,173.145,27.016,154.877
C08582=1069.851,137.188,425.122,173.144,27.014,154.876
C08583=1069.845,136.940,425.142,173.142,27.011,154.876
C08584=1069.839,136.690,425.163,173.141,27.008,154.876
C08585=1069.834,136.441,425.183,173.138,27.006,154.875
C08586=1069.828,136.192,425.203,173.137,27.003,154.875
C08587=1069.822,135.943,425.225,173.135,27.000,154.875
C08588=1069.816,135.694,425.245,173.134,26.997,154.874
C08589=1069.810,135.445,425.265,173.131,26.995,154.874
C08590=1069.804,135.196,425.285,173.130,26.992,154.874
C08591=1069.799,134.947,425.306,173.128,26.989,154.873
C08592=1069.793,134.697,425.326,173.127,26.986,154.873
C08593=1069.787,134.448,425.347,173.125,26.984,154.872
C08594=1069.781,134.199,425.367,173.123,26.981,154.872
C08595=1069.776,133.950,425.387,173.122,26.978,154.872
C08596=1069.771,133.701,425.408,173.120,26.975,154.871
C08597=1069.764,133.451,425.428,173.118,26.973,154.871
C08598=1069.759,133.202,425.449,173.116,26.970,154.871
C08599=1069.753,132.954,425.469,173.115,26.967,154.870
C08600=1069.748,132.704,425.489,173.113,26.964,154.870
C08601=1069.742,132.456,425.509,173.112,26.962,154.869
C08602=1069.736,132.207,425.530,173.109,26.959,154.869
C08603=1069.730,131.957,425.550,173.108,26.956,154.869
C08604=1069.724,131.708,425.570,173.106,26.954,154.868
C08605=1069.719,131.459,425.591,173.105,26.951,154.868
C08606=1069.713,131.210,425.610,173.103,26.948,154.868
C08607=1069.707,130.961,425.630,173.101,26.945,154.867
C08608=1069.701,130.711,425.651,173.099,26.943,154.867
C08609=1069.695,130.462,425.671,173.098,26.940,154.867
C08610=1069.689,130.213,425.691,173.096,26.938,154.866
C08611=1069.683,129.965,425.711,173.094,26.935,154.866
C08612=1069.678,129.715,425.731,173.092,26.932,154.865
C08613=1069.671,129.466,425.752,173.091,26.929,154.865
C08614=1069.666,129.216,425.771,173.089,26.927,154.865
C08615=1069.660,128.967,425.791,173.088,26.924,154.864
C08616=1069.654,128.719,425.811,173.086,26.921,154.864
C08617=1069.648,128.470,425.831,173.084,26.919,154.864
C08618=1069.642,128.221,425.851,173.083,26.916,154.863
C08619=1069.637,127.970,425.871,173.081,26.913,154.863
C08620=1069.631,127.722,425.891,173.080,26.911,154.863
C08621=1069.625,127.473,425.911,173.077,26.908,154.862
C08622=1069.618,127.190,425.934,173.076,26.905,154.862
C08623=1069.612,126.907,425.956,173.073,26.902,154.861
C08624=1069.605,126.624,425.979,173.072,26.899,154.861
C08625=1069.599,126.342,426.002,173.070,26.896,154.861
C08626=1069.592,126.092,426.022,173.068,26.894,154.860
C08627=1069.587,125.843,426.042,173.067,26.891,154.860
C08628=1069.581,125.594,426.062,173.065,26.888,154.859
C08629=1069.575,125.345,426.082,173.064,26.885,154.859
C08630=1069.570,125.095,426.101,173.061,26.883,154.859
C08631=1069.564,124.846,426.121,173.060,26.880,154.858
C08632=1069.558,124.598,426.141,173.058,26.877,154.858
C08633=1069.553,124.348,426.161,173.057,26.875,154.858
C08634=1069.547,124.099,426.181,173.055,26.872,154.857
C08635=1069.541,123.850,426.201,173.054,26.869,154.857
C08636=1069.535,123.601,426.220,173.052,26.866,154.857
C08637=1069.528,123.351,426.241,173.050,26.864,154.856
C08638=1069.523,123.102,426.261,173.049,26.861,154.856
C08639=1069.517,122.853,426.280,173.047,26.858,154.855
C08640=1069.512,122.604,426.300,173.046,26.855,154.855
C08641=1069.506,122.354,426.320,173.043,26.853,154.855
C08642=1069.500,122.106,426.340,173.042,26.850,154.854
C08643=1069.494,121.857,426.359,173.040,26.847,154.854
C08644=1069.489,121.607,426.379,173.039,26.844,154.854
C08645=1069.483,121.358,426.399,173.037,26.842,154.853
C08646=1069.477,121.109,426.419,173.036,26.839,154.853
C08647=1069.471,120.860,426.438,173.033,26.836,154.853
C08648=1069.466,120.611,426.458,173.032,26.833,154.852
C08649=1069.460,120.362,426.478,173.031,26.831,154.852
C08650=1069.455,120.112,426.498,173.029,26.828,154.851
C08651=1069.449,119.863,426.517,173.028,26.826,154.851
C08652=1069.443,119.614,426.537,173.026,26.823,154.851
C08653=1069.437,119.365,426.557,173.024,26.820,154.850
C08654=1069.431,119.116,426.576,173.022,26.817,154.850
C08655=1069.425,118.867,426.596,173.021,26.815,154.850
C08656=1069.420,118.617,426.616,173.019,26.812,154.849
C08657=1069.414,118.368,426.636,173.018,26.809,154.849
C08658=1069.409,118.119,426.655,173.016,26.806,154.848
C08659=1069.403,117.871,426.675,173.015,26.803,154.848
C08660=1069.398,117.621,426.694,173.012,26.801,154.848
C08661=1069.392,117.372,426.713,173.011,26.798,154.847
C08662=1069.386,117.123,426.733,173.010,26.795,154.847
C08663=1069.380,116.874,426.752,173.008,26.792,154.846
C08664=1069.375,116.624,426.773,173.007,26.790,154.846
C08665=1069.369,116.375,426.792,173.005,26.787,154.846
C08666=1069.364,116.126,426.811,173.003,26.784,154.845
C08667=1069.358,115.877,426.831,173.001,26.781,154.845
C08668=1069.352,115.627,426.850,173.000,26.779,154.845
C08669=1069.346,115.378,426.870,172.998,26.776,154.844
C08670=1069.341,115.130,426.889,172.997,26.773,154.844
C08671=1069.335,114.880,426.909,172.995,26.771,154.843
C08672=1069.329,114.631,426.928,172.994,26.768,154.843
C08673=1069.324,114.382,426.948,172.993,26.765,154.843
C08674=1069.318,114.132,426.968,172.990,26.762,154.842
C08675=1069.312,113.883,426.986,172.989,26.759,154.842
C08676=1069.306,113.634,427.006,172.987,26.757,154.842
C08677=1069.300,113.385,427.025,172.986,26.754,154.841
C08678=1069.295,113.136,427.045,172.984,26.751,154.841
C08679=1069.289,112.886,427.064,172.983,26.748,154.840
C08680=1069.283,112.637,427.084,172.981,26.746,154.840
C08681=1069.278,112.389,427.103,172.979,26.743,154.840
C08682=1069.272,112.139,427.122,172.978,26.740,154.839
C08683=1069.266,111.890,427.141,172.976,26.737,154.839
C08684=1069.260,111.641,427.161,172.975,26.735,154.839
C08685=1069.254,111.392,427.180,172.973,26.732,154.838
C08686=1069.248,111.109,427.202,172.971,26.729,154.838
C08687=1069.241,110.825,427.224,172.969,26.726,154.837
C08688=1069.235,110.543,427.246,172.968,26.723,154.837
C08689=1069.228,110.259,427.267,172.966,26.720,154.837
C08690=1069.222,110.010,427.286,172.964,26.717,154.836
C08691=1069.216,109.761,427.305,172.963,26.715,154.836
C08692=1069.210,109.512,427.324,172.961,26.712,154.835
C08693=1069.204,109.263,427.344,172.960,26.709,154.835
C08694=1069.199,109.014,427.363,172.958,26.706,154.835
C08695=1069.192,108.765,427.382,172.957,26.704,154.834
C08696=1069.187,108.515,427.401,172.954,26.701,154.834
C08697=1069.181,108.266,427.420,172.953,26.698,154.834
C08698=1069.176,108.017,427.439,172.952,26.695,154.833
C08699=1069.169,107.768,427.458,172.950,26.693,154.833
C08700=1069.164,107.518,427.477,172.949,26.690,154.833
C08701=1069.158,107.269,427.496,172.947,26.688,154.832
C08702=1069.152,107.020,427.516,172.946,26.685,154.832
C08703=1069.146,106.770,427.534,172.944,26.682,154.831
C08704=1069.141,106.522,427.553,172.942,26.679,154.831
C08705=1069.135,106.272,427.572,172.940,26.677,154.831
C08706=1069.129,106.023,427.591,172.939,26.674,154.830
C08707=1069.123,105.774,427.610,172.937,26.671,154.830
C08708=1069.117,105.524,427.629,172.936,26.669,154.830
C08709=1069.112,105.275,427.649,172.935,26.666,154.829
C08710=1069.106,105.026,427.667,172.933,26.663,154.829
C08711=1069.100,104.777,427.686,172.932,26.661,154.828
C08712=1069.094,104.528,427.706,172.930,26.658,154.828
C08713=1069.088,104.278,427.724,172.929,26.655,154.828
C08714=1069.083,104.030,427.743,172.926,26.652,154.827
C08715=1069.077,103.780,427.762,172.925,26.650,154.827
C08716=1069.071,103.531,427.781,172.923,26.647,154.827
C08717=1069.065,103.282,427.800,172.922,26.644,154.826
C08718=1069.059,103.032,427.819,172.921,26.641,154.826
C08719=1069.054,102.784,427.838,172.919,26.638,154.825
C08720=1069.048,102.534,427.857,172.918,26.636,154.825
C08721=1069.043,102.284,427.875,172.916,26.633,154.825
C08722=1069.037,102.035,427.895,172.915,26.631,154.824
C08723=1069.031,101.787,427.913,172.913,26.628,154.824
C08724=1069.025,101.537,427.932,172.911,26.625,154.824
C08725=1069.019,101.288,427.951,172.910,26.622,154.823
C08726=1069.014,101.039,427.970,172.908,26.619,154.823
C08727=1069.008,100.790,427.989,172.907,26.617,154.822
C08728=1069.002,100.540,428.007,172.905,26.614,154.822
C08729=1068.996,100.291,428.026,172.904,26.612,154.822
C08730=1068.990,100.041,428.045,172.902,26.609,154.821
C08731=1068.984,99.793,428.063,172.901,26.606,154.821
C08732=1068.978,99.544,428.082,172.899,26.603,154.821
C08733=1068.972,99.294,428.100,172.898,26.601,154.820
C08734=1068.967,99.044,428.120,172.896,26.598,154.820
C08735=1068.961,98.796,428.138,172.894,26.595,154.819
C08736=1068.955,98.547,428.157,172.892,26.593,154.819
C08737=1068.949,98.297,428.175,172.891,26.590,154.819
C08738=1068.944,98.048,428.194,172.890,26.587,154.818
C08739=1068.937,97.799,428.213,172.888,26.584,154.818
C08740=1068.932,97.550,428.232,172.887,26.582,154.818
C08741=1068.926,97.300,428.250,172.885,26.579,154.817
C08742=1068.920,97.051,428.268,172.884,26.576,154.817
C08743=1068.914,96.802,428.287,172.882,26.573,154.817
C08744=1068.908,96.552,428.305,172.881,26.571,154.816
C08745=1068.903,96.304,428.324,172.879,26.568,154.816
C08746=1068.896,96.054,428.343,172.878,26.565,154.815
C08747=1068.891,95.804,428.361,172.877,26.563,154.815
C08748=1068.885,95.556,428.379,172.874,26.560,154.815
C08749=1068.879,95.307,428.398,172.873,26.557,154.814
C08750=1068.872,95.024,428.419,172.871,26.554,154.814
C08751=1068.866,94.741,428.440,172.870,26.551,154.813
C08752=1068.859,94.458,428.461,172.868,26.548,154.813
C08753=1068.853,94.175,428.482,172.866,26.545,154.813
C08754=1068.847,93.925,428.501,172.865,26.542,154.812
C08755=1068.841,93.676,428.519,172.863,26.539,154.812
C08756=1068.835,93.427,428.537,172.862,26.537,154.811
C08757=1068.830,93.177,428.556,172.861,26.534,154.811
C08758=1068.824,92.928,428.574,172.859,26.531,154.811
C08759=1068.818,92.679,428.593,172.858,26.529,154.810
C08760=1068.812,92.430,428.612,172.855,26.525,154.810
C08761=1068.807,92.181,428.629,172.854,26.523,154.810
C08762=1068.801,91.931,428.648,172.852,26.520,154.809
C08763=1068.795,91.682,428.666,172.851,26.518,154.809
C08764=1068.789,91.433,428.685,172.850,26.515,154.809
C08765=1068.784,91.183,428.703,172.848,26.512,154.808
C08766=1068.778,90.935,428.721,172.847,26.509,154.808
C08767=1068.772,90.685,428.739,172.845,26.506,154.807
C08768=1068.766,90.436,428.759,172.844,26.504,154.807
C08769=1068.760,90.186,428.776,172.842,26.501,154.807
C08770=1068.754,89.937,428.795,172.841,26.498,154.806
C08771=1068.748,89.688,428.813,172.839,26.496,154.806
C08772=1068.742,89.439,428.830,172.838,26.493,154.806
C08773=1068.736,89.189,428.849,172.837,26.490,154.805
C08774=1068.731,88.940,428.867,172.835,26.488,154.805
C08775=1068.725,88.691,428.886,172.834,26.485,154.804
C08776=1068.719,88.441,428.904,172.832,26.482,154.804
C08777=1068.713,88.192,428.921,172.830,26.479,154.804
C08778=1068.707,87.943,428.940,172.828,26.477,154.803
C08779=1068.701,87.694,428.958,172.827,26.474,154.803
C08780=1068.695,87.445,428.976,172.825,26.471,154.803
C08781=1068.689,87.195,428.995,172.824,26.468,154.802
C08782=1068.684,86.946,429.012,172.823,26.466,154.802
C08783=1068.677,86.697,429.031,172.821,26.463,154.802
C08784=1068.672,86.448,429.048,172.820,26.461,154.801
C08785=1068.666,86.198,429.066,172.818,26.458,154.801
C08786=1068.659,85.949,429.085,172.817,26.455,154.800
C08787=1068.654,85.700,429.103,172.815,26.453,154.800
C08788=1068.648,85.450,429.121,172.814,26.450,154.800
C08789=1068.643,85.201,429.139,172.812,26.447,154.799
C08790=1068.636,84.952,429.157,172.811,26.445,154.799
C08791=1068.631,84.703,429.175,172.810,26.442,154.799
C08792=1068.625,84.453,429.193,172.808,26.439,154.798
C08793=1068.619,84.204,429.211,172.807,26.436,154.798
C08794=1068.613,83.955,429.229,172.805,26.434,154.797
C08795=1068.607,83.706,429.247,172.804,26.431,154.797
C08796=1068.601,83.456,429.265,172.802,26.428,154.797
C08797=1068.595,83.207,429.283,172.801,26.425,154.796
C08798=1068.590,82.957,429.301,172.799,26.423,154.796
C08799=1068.584,82.708,429.319,172.797,26.420,154.796
C08800=1068.578,82.459,429.337,172.796,26.417,154.795
C08801=1068.573,82.210,429.354,172.794,26.414,154.795
C08802=1068.566,81.960,429.373,172.793,26.411,154.794
C08803=1068.561,81.711,429.391,172.791,26.409,154.794
C08804=1068.555,81.462,429.409,172.790,26.406,154.794
C08805=1068.549,81.213,429.426,172.789,26.403,154.793
C08806=1068.543,80.963,429.444,172.787,26.401,154.793
C08807=1068.538,80.714,429.462,172.786,26.398,154.792
C08808=1068.531,80.465,429.480,172.784,26.395,154.792
C08809=1068.526,80.216,429.498,172.783,26.393,154.792
C08810=1068.520,79.966,429.516,172.782,26.390,154.791
C08811=1068.514,79.717,429.533,172.780,26.387,154.791
C08812=1068.509,79.468,429.552,172.779,26.384,154.791
C08813=1068.503,79.218,429.569,172.777,26.382,154.790
C08814=1068.496,78.935,429.590,172.776,26.378,154.790
C08815=1068.489,78.653,429.609,172.774,26.375,154.789
C08816=1068.483,78.369,429.630,172.772,26.372,154.789
C08817=1068.476,78.086,429.650,172.771,26.369,154.789
C08818=1068.470,77.837,429.667,172.769,26.367,154.788
C08819=1068.464,77.588,429.685,172.768,26.364,154.788
C08820=1068.459,77.339,429.703,172.767,26.361,154.787
C08821=1068.453,77.089,429.721,172.765,26.358,154.787
C08822=1068.447,76.840,429.738,172.764,26.356,154.787
C08823=1068.441,76.590,429.756,172.762,26.353,154.786
C08824=1068.435,76.341,429.773,172.761,26.350,154.786
C08825=1068.429,76.092,429.791,172.758,26.348,154.786
C08826=1068.423,75.843,429.809,172.757,26.345,154.785
C08827=1068.418,75.594,429.826,172.756,26.342,154.785
C08828=1068.412,75.344,429.844,172.754,26.339,154.785
C08829=1068.406,75.095,429.862,172.753,26.337,154.784
C08830=1068.399,74.845,429.879,172.751,26.334,154.784
C08831=1068.394,74.596,429.897,172.750,26.331,154.783
C08832=1068.388,74.347,429.914,172.748,26.328,154.783
C08833=1068.382,74.097,429.932,172.747,26.326,154.783
C08834=1068.376,73.848,429.950,172.746,26.323,154.782
C08835=1068.370,73.598,429.967,172.744,26.320,154.782
C08836=1068.364,73.349,429.984,172.743,26.317,154.782
C08837=1068.359,73.100,430.002,172.741,26.315,154.781
C08838=1068.353,72.851,430.020,172.740,26.312,154.781
C08839=1068.347,72.602,430.037,172.738,26.309,154.780
C08840=1068.342,72.353,430.055,172.737,26.307,154.780
C08841=1068.335,72.103,430.072,172.736,26.304,154.780
C08842=1068.329,71.854,430.090,172.734,26.301,154.779
C08843=1068.324,71.604,430.107,172.733,26.299,154.779
C08844=1068.318,71.355,430.124,172.731,26.296,154.779
C08845=1068.312,71.106,430.141,172.730,26.293,154.778
C08846=1068.306,70.856,430.159,172.728,26.291,154.778
C08847=1068.300,70.607,430.177,172.727,26.288,154.777
C08848=1068.295,70.358,430.194,172.726,26.285,154.777
C08849=1068.288,70.108,430.211,172.724,26.282,154.777
C08850=1068.283,69.859,430.229,172.723,26.280,154.776
C08851=1068.277,69.610,430.246,172.721,26.277,154.776
C08852=1068.270,69.361,430.264,172.720,26.274,154.776
C08853=1068.265,69.111,430.280,172.719,26.271,154.775
C08854=1068.259,68.862,430.298,172.717,26.269,154.775
C08855=1068.253,68.612,430.315,172.716,26.266,154.775
C08856=1068.247,68.363,430.333,172.714,26.263,154.774
C08857=1068.242,68.114,430.350,172.713,26.260,154.774
C08858=1068.235,67.864,430.367,172.711,26.258,154.773
C08859=1068.229,67.615,430.385,172.710,26.255,154.773
C08860=1068.224,67.366,430.402,172.709,26.252,154.773
C08861=1068.217,67.116,430.419,172.707,26.250,154.772
C08862=1068.212,66.867,430.436,172.706,26.247,154.772
C08863=1068.206,66.618,430.453,172.704,26.244,154.772
C08864=1068.200,66.368,430.471,172.703,26.241,154.771
C08865=1068.194,66.119,430.488,172.701,26.239,154.771
C08866=1068.188,65.870,430.504,172.700,26.236,154.770
C08867=1068.182,65.620,430.522,172.699,26.233,154.770
C08868=1068.176,65.371,430.539,172.697,26.231,154.770
C08869=1068.171,65.121,430.556,172.696,26.228,154.769
C08870=1068.165,64.872,430.574,172.694,26.225,154.769
C08871=1068.158,64.623,430.591,172.693,26.223,154.769
C08872=1068.153,64.373,430.608,172.692,26.220,154.768
C08873=1068.147,64.125,430.625,172.690,26.217,154.768
C08874=1068.141,63.874,430.642,172.689,26.215,154.768
C08875=1068.135,63.626,430.659,172.687,26.212,154.767
C08876=1068.129,63.376,430.675,172.686,26.209,154.767
C08877=1068.123,63.126,430.693,172.684,26.207,154.766
C08878=1068.116,62.844,430.712,172.682,26.203,154.766
C08879=1068.109,62.561,430.732,172.681,26.201,154.766
C08880=1068.102,62.277,430.751,172.679,26.198,154.765
C08881=1068.096,61.995,430.770,172.678,26.195,154.765
C08882=1068.089,61.746,430.787,172.677,26.192,154.764
C08883=1068.083,61.496,430.804,172.675,26.189,154.764
C08884=1068.077,61.247,430.821,172.674,26.187,154.764
C08885=1068.071,60.997,430.837,172.672,26.184,154.763
C08886=1068.065,60.748,430.855,172.671,26.182,154.763
C08887=1068.059,60.498,430.872,172.669,26.179,154.763
C08888=1068.053,60.250,430.889,172.668,26.176,154.762
C08889=1068.048,60.000,430.905,172.666,26.174,154.762
C08890=1068.041,59.750,430.922,172.665,26.171,154.762
C08891=1068.035,59.501,430.939,172.664,26.168,154.761
C08892=1068.030,59.251,430.956,172.661,26.165,154.761
C08893=1068.024,59.003,430.973,172.660,26.162,154.761
C08894=1068.017,58.753,430.990,172.658,26.160,154.760
C08895=1068.011,58.504,431.006,172.657,26.157,154.760
C08896=1068.006,58.254,431.023,172.656,26.154,154.760
C08897=1068.000,58.005,431.040,172.654,26.152,154.759
C08898=1067.993,57.756,431.057,172.653,26.149,154.759
C08899=1067.988,57.506,431.074,172.651,26.146,154.758
C08900=1067.981,57.257,431.091,172.650,26.144,154.758
C08901=1067.975,57.008,431.107,172.648,26.141,154.758
C08902=1067.970,56.758,431.124,172.647,26.138,154.757
C08903=1067.963,56.509,431.141,172.646,26.136,154.757
C08904=1067.957,56.259,431.157,172.644,26.133,154.757
C08905=1067.952,56.010,431.174,172.643,26.130,154.756
C08906=1067.946,55.761,431.191,172.642,26.128,154.756
C08907=1067.940,55.512,431.208,172.641,26.125,154.755
C08908=1067.934,55.262,431.224,172.639,26.123,154.755
C08909=1067.928,55.012,431.241,172.638,26.120,154.755
C08910=1067.922,54.763,431.258,172.637,26.117,154.754
C08911=1067.916,54.514,431.274,172.635,26.115,154.754
C08912=1067.911,54.264,431.291,172.634,26.112,154.754
C08913=1067.904,54.015,431.308,172.632,26.109,154.753
C08914=1067.898,53.766,431.324,172.631,26.106,154.753
C08915=1067.892,53.516,431.341,172.630,26.104,154.753
C08916=1067.887,53.266,431.358,172.628,26.101,154.752
C08917=1067.880,53.018,431.375,172.627,26.098,154.752
C08918=1067.875,52.768,431.391,172.625,26.096,154.752
C08919=1067.869,52.519,431.407,172.624,26.093,154.751
C08920=1067.863,52.269,431.424,172.623,26.090,154.751
C08921=1067.857,52.020,431.440,172.621,26.088,154.751
C08922=1067.851,51.771,431.457,172.620,26.085,154.750
C08923=1067.845,51.522,431.474,172.618,26.082,154.750
C08924=1067.839,51.271,431.491,172.617,26.079,154.749
C08925=1067.833,51.022,431.507,172.615,26.077,154.749
C08926=1067.827,50.773,431.523,172.614,26.074,154.749
C08927=1067.821,50.524,431.540,172.613,26.071,154.748
C08928=1067.816,50.274,431.557,172.611,26.068,154.748
C08929=1067.810,50.025,431.573,172.610,26.066,154.748
C08930=1067.804,49.776,431.590,172.608,26.063,154.747
C08931=1067.798,49.526,431.606,172.607,26.060,154.747
C08932=1067.793,49.277,431.623,172.606,26.057,154.746
C08933=1067.787,49.027,431.639,172.604,26.055,154.746
C08934=1067.781,48.778,431.655,172.603,26.052,154.746
C08935=1067.775,48.529,431.672,172.601,26.049,154.745
C08936=1067.769,48.280,431.689,172.600,26.047,154.745
C08937=1067.764,48.030,431.705,172.599,26.044,154.745
C08938=1067.758,47.781,431.722,172.597,26.041,154.744
C08939=1067.752,47.532,431.738,172.596,26.038,154.744
C08940=1067.746,47.282,431.754,172.594,26.036,154.744
C08941=1067.740,47.033,431.770,172.593,26.033,154.743
C08942=1067.731,46.649,431.796,172.591,26.029,154.743
C08943=1067.722,46.265,431.822,172.589,26.025,154.742
C08944=1067.713,45.881,431.847,172.587,26.020,154.741
C08945=1067.705,45.498,431.872,172.585,26.016,154.741
C08946=1067.699,45.248,431.888,172.583,26.014,154.740
C08947=1067.693,44.999,431.904,172.582,26.011,154.740
C08948=1067.687,44.750,431.921,172.581,26.008,154.740
C08949=1067.681,44.500,431.937,172.579,26.006,154.739
C08950=1067.676,44.251,431.954,172.578,26.003,154.739
C08951=1067.670,44.001,431.970,172.576,26.000,154.739
C08952=1067.664,43.752,431.986,172.575,25.997,154.738
C08953=1067.658,43.502,432.002,172.573,25.995,154.738
C08954=1067.652,43.253,432.018,172.572,25.992,154.738
C08955=1067.646,43.003,432.034,172.571,25.989,154.737
C08956=1067.640,42.754,432.050,172.569,25.987,154.737
C08957=1067.634,42.505,432.067,172.568,25.984,154.736
C08958=1067.628,42.255,432.083,172.566,25.981,154.736
C08959=1067.622,42.006,432.099,172.565,25.979,154.736
C08960=1067.616,41.756,432.115,172.564,25.976,154.735
C08961=1067.610,41.507,432.132,172.562,25.973,154.735
C08962=1067.605,41.257,432.147,172.561,25.970,154.735
C08963=1067.599,41.008,432.164,172.559,25.968,154.734
C08964=1067.593,40.758,432.180,172.558,25.965,154.734
C08965=1067.586,40.509,432.195,172.557,25.962,154.734
C08966=1067.577,40.110,432.222,172.555,25.958,154.733
C08967=1067.568,39.713,432.248,172.552,25.954,154.732
C08968=1067.558,39.314,432.273,172.549,25.949,154.732
C08969=1067.549,38.916,432.298,172.547,25.945,154.731
C08970=1067.543,38.667,432.315,172.546,25.943,154.731
C08971=1067.537,38.417,432.331,172.545,25.940,154.731
C08972=1067.532,38.167,432.346,172.543,25.937,154.730
C08973=1067.526,37.918,432.363,172.542,25.934,154.730
C08974=1067.519,37.669,432.378,172.540,25.932,154.730
C08975=1067.513,37.419,432.394,172.539,25.929,154.729
C08976=1067.507,37.170,432.410,172.538,25.926,154.729
C08977=1067.502,36.920,432.426,172.536,25.924,154.728
C08978=1067.495,36.671,432.442,172.535,25.921,154.728
C08979=1067.489,36.421,432.457,172.533,25.918,154.728
C08980=1067.483,36.172,432.474,172.532,25.915,154.727
C08981=1067.477,35.922,432.490,172.530,25.913,154.727
C08982=1067.471,35.673,432.506,172.529,25.910,154.727
C08983=1067.465,35.423,432.521,172.528,25.908,154.726
C08984=1067.460,35.175,432.537,172.526,25.905,154.726
C08985=1067.454,34.925,432.553,172.525,25.903,154.726
C08986=1067.447,34.676,432.568,172.523,25.900,154.725
C08987=1067.441,34.426,432.585,172.522,25.897,154.725
C08988=1067.436,34.176,432.600,172.522,25.895,154.725
C08989=1067.430,33.927,432.616,172.520,25.892,154.724
C08990=1067.423,33.678,432.632,172.519,25.890,154.724
C08991=1067.417,33.428,432.648,172.517,25.887,154.724
C08992=1067.411,33.179,432.664,172.516,25.884,154.723
C08993=1067.406,32.929,432.679,172.514,25.882,154.723
C08994=1067.400,32.680,432.695,172.513,25.879,154.723
C08995=1067.394,32.431,432.711,172.512,25.876,154.722
C08996=1067.388,32.181,432.726,172.510,25.874,154.722
C08997=1067.381,31.932,432.742,172.509,25.871,154.721
C08998=1067.376,31.682,432.758,172.507,25.868,154.721
C08999=1067.370,31.433,432.774,172.506,25.866,154.721
C09000=1067.363,31.183,432.789,172.505,25.863,154.721
C09001=1067.358,30.935,432.805,172.503,25.860,154.720
C09002=1067.351,30.651,432.823,172.501,25.857,154.720
C09003=1067.344,30.367,432.840,172.500,25.854,154.719
C09004=1067.338,30.084,432.858,172.498,25.851,154.719
C09005=1067.331,29.801,432.876,172.497,25.848,154.719
C09006=1067.325,29.551,432.891,172.496,25.846,154.718
C09007=1067.319,29.302,432.908,172.494,25.843,154.718
C09008=1067.313,29.052,432.922,172.493,25.840,154.718
C09009=1067.308,28.804,432.938,172.491,25.838,154.717
C09010=1067.302,28.554,432.954,172.490,25.835,154.717
C09011=1067.295,28.305,432.970,172.489,25.832,154.716
C09012=1067.290,28.055,432.985,172.487,25.830,154.716
C09013=1067.283,27.806,433.001,172.486,25.827,154.716
C09014=1067.277,27.556,433.016,172.484,25.824,154.715
C09015=1067.272,27.306,433.031,172.483,25.822,154.715
C09016=1067.266,27.057,433.047,172.481,25.819,154.715
C09017=1067.260,26.807,433.063,172.480,25.817,154.714
C09018=1067.253,26.558,433.078,172.479,25.814,154.714
C09019=1067.248,26.308,433.094,172.477,25.811,154.714
C09020=1067.242,26.059,433.108,172.476,25.809,154.713
C09021=1067.236,25.810,433.125,172.474,25.806,154.713
C09022=1067.229,25.560,433.140,172.473,25.803,154.713
C09023=1067.224,25.310,433.155,172.472,25.801,154.712
C09024=1067.217,25.061,433.171,172.470,25.798,154.712
C09025=1067.212,24.812,433.186,172.469,25.796,154.712
C09026=1067.206,24.562,433.201,172.467,25.793,154.711
C09027=1067.200,24.313,433.217,172.466,25.791,154.711
C09028=1067.193,24.063,433.232,172.465,25.788,154.711
C09029=1067.188,23.813,433.248,172.463,25.785,154.710
C09030=1067.182,23.565,433.263,172.462,25.783,154.710
C09031=1067.175,23.315,433.278,172.460,25.780,154.710
C09032=1067.170,23.065,433.294,172.459,25.777,154.709
C09033=1067.163,22.816,433.308,172.458,25.774,154.709
C09034=1067.158,22.567,433.324,172.456,25.772,154.709
C09035=1067.151,22.317,433.339,172.455,25.769,154.708
C09036=1067.146,22.068,433.355,172.453,25.767,154.708
C09037=1067.140,21.819,433.369,172.452,25.764,154.708
C09038=1067.134,21.569,433.386,172.450,25.762,154.707
C09039=1067.128,21.320,433.401,172.449,25.759,154.707
C09040=1067.122,21.070,433.416,172.448,25.756,154.707
C09041=1067.116,20.821,433.431,172.446,25.754,154.706
C09042=1067.111,20.571,433.446,172.445,25.751,154.706
C09043=1067.104,20.322,433.462,172.443,25.748,154.706
C09044=1067.098,20.072,433.477,172.442,25.746,154.705
C09045=1067.093,19.823,433.492,172.441,25.743,154.705
C09046=1067.086,19.573,433.507,172.439,25.741,154.705
C09047=1067.080,19.323,433.522,172.438,25.738,154.704
C09048=1067.075,19.074,433.537,172.436,25.736,154.704
C09049=1067.068,18.825,433.553,172.435,25.733,154.704
C09050=1067.062,18.575,433.568,172.434,25.731,154.703
C09051=1067.056,18.325,433.583,172.433,25.728,154.703
C09052=1067.050,18.077,433.598,172.432,25.725,154.703
C09053=1067.044,17.827,433.613,172.430,25.723,154.702
C09054=1067.038,17.577,433.628,172.429,25.720,154.702
C09055=1067.032,17.328,433.643,172.427,25.718,154.702
C09056=1067.026,17.078,433.658,172.426,25.715,154.701
C09057=1067.020,16.828,433.673,172.424,25.713,154.701
C09058=1067.014,16.580,433.689,172.423,25.710,154.701
C09059=1067.008,16.330,433.704,172.422,25.707,154.700
C09060=1067.002,16.081,433.719,172.420,25.705,154.700
C09061=1066.996,15.831,433.734,172.419,25.702,154.700
C09062=1066.990,15.582,433.749,172.418,25.699,154.699
C09063=1066.984,15.332,433.764,172.416,25.697,154.699
C09064=1066.979,15.083,433.779,172.415,25.694,154.699
C09065=1066.972,14.833,433.794,172.413,25.692,154.698
C09066=1066.965,14.551,433.811,172.412,25.689,154.698
C09067=1066.959,14.269,433.827,172.410,25.686,154.698
C09068=1066.952,13.987,433.845,172.408,25.683,154.697
C09069=1066.945,13.705,433.861,172.407,25.680,154.697
C09070=1066.939,13.456,433.876,172.405,25.678,154.697
C09071=1066.933,13.207,433.891,172.404,25.675,154.696
C09072=1066.926,12.957,433.906,172.403,25.673,154.696
C09073=1066.920,12.708,433.920,172.401,25.670,154.696
C09074=1066.914,12.458,433.935,172.400,25.668,154.695
C09075=1066.909,12.208,433.950,172.398,25.665,154.695
C09076=1066.903,11.959,433.965,172.397,25.662,154.695
C09077=1066.897,11.709,433.980,172.395,25.660,154.694
C09078=1066.890,11.459,433.995,172.394,25.657,154.694
C09079=1066.884,11.211,434.009,172.393,25.655,154.694
C09080=1066.878,10.961,434.024,172.391,25.653,154.693
C09081=1066.872,10.712,434.039,172.390,25.650,154.693
C09082=1066.866,10.462,434.054,172.388,25.647,154.693
C09083=1066.860,10.213,434.069,172.387,25.645,154.692
C09084=1066.854,9.963,434.082,172.386,25.642,154.692
C09085=1066.848,9.713,434.097,172.384,25.640,154.692
C09086=1066.841,9.464,434.112,172.383,25.637,154.692
C09087=1066.835,9.215,434.127,172.381,25.635,154.691
C09088=1066.829,8.965,434.142,172.380,25.632,154.691
C09089=1066.823,8.716,434.156,172.378,25.630,154.691
C09090=1066.817,8.466,434.171,172.377,25.627,154.690
C09091=1066.812,8.216,434.186,172.376,25.625,154.690
C09092=1066.806,7.967,434.201,172.374,25.622,154.690
C09093=1066.799,7.717,434.216,172.373,25.619,154.689
C09094=1066.794,7.468,434.230,172.371,25.617,154.689
C09095=1066.788,7.218,434.245,172.370,25.615,154.689
C09096=1066.782,6.969,434.259,172.369,25.612,154.688
C09097=1066.775,6.719,434.274,172.367,25.610,154.688
C09098=1066.770,6.471,434.289,172.366,25.607,154.688
C09099=1066.764,6.220,434.303,172.364,25.604,154.687
C09100=1066.757,5.971,434.318,172.363,25.602,154.687
C09101=1066.751,5.722,434.332,172.361,25.600,154.687
C09102=1066.745,5.472,434.347,172.360,25.597,154.686
C09103=1066.740,5.222,434.361,172.359,25.594,154.686
C09104=1066.733,4.973,434.376,172.357,25.592,154.686
